  MoveL 635 to (33.53, 138.59, 49.77) mm, rotated rx 110.14 ry 0 rz -13.26 deg; joints [126.944, -22.767, 36.217, -107.187, 38.986, 156.564, 25, 13.26]
  MoveL 636 to (34.49, 138.1, 50.45) mm, rotated rx 110.14 ry 0 rz -13.26 deg; joints [126.986, -22.796, 36.22, -107.13, 39.017, 156.503, 25, 13.26]
  MoveL 637 to (34.94, 137.59, 51.53) mm, rotated rx 110.14 ry 0 rz -13.26 deg; joints [127.026, -22.799, 36.192, -107.072, 39.045, 156.439, 25, 13.26]
  MoveL 638 to (34.99, 137.43, 51.91) mm, rotated rx 110.29 ry 0 rz -13.29 deg; joints [127.07, -22.764, 36.12, -107.001, 39.075, 156.207, 25, 13.293]
  MoveL 639 to (34.9, 137.09, 52.87) mm, rotated rx 110.29 ry 0 rz -13.29 deg; joints [127.093, -22.746, 36.081, -106.964, 39.09, 156.166, 25, 13.293]
  MoveL 640 to (34.24, 136.43, 54.94) mm, rotated rx 111.13 ry 0 rz -13.09 deg; joints [127.332, -22.556, 35.689, -106.59, 39.255, 154.912, 25, 13.093]
  MoveL 641 to (34.22, 136.45, 54.91) mm, rotated rx 112.01 ry 0 rz -13.37 deg; joints [127.511, -22.368, 35.349, -106.31, 39.379, 153.728, 25, 13.374]
  MoveL 642 to (35.06, 135.89, 55.75) mm, rotated rx 112.35 ry 0 rz -13.76 deg; joints [127.61, -22.288, 35.19, -106.163, 39.45, 153.224, 25, 13.758]
  MoveL 643 to (35.03, 135.9, 55.76) mm, rotated rx 112.58 ry 0 rz -14.72 deg; joints [127.605, -22.149, 35.037, -106.15, 39.441, 152.972, 25, 14.719]
  MoveL 644 to (36.59, 135.66, 55.37) mm, rotated rx 112.43 ry 0 rz -15.36 deg; joints [127.559, -22.187, 35.111, -106.218, 39.408, 153.203, 25, 15.358]
  MoveL 645 to (37.62, 135.39, 55.32) mm, rotated rx 112.43 ry 0 rz -15.36 deg; joints [127.584, -22.23, 35.142, -106.19, 39.428, 153.175, 25, 15.358]
  MoveL 646 to (37.97, 135.27, 55.38) mm, rotated rx 112.45 ry 0 rz -15.51 deg; joints [127.591, -22.225, 35.131, -106.18, 39.433, 153.14, 25, 15.509]
  MoveL 647 to (38.54, 135.04, 55.55) mm, rotated rx 112.45 ry 0 rz -15.51 deg; joints [127.61, -22.245, 35.141, -106.156, 39.448, 153.115, 25, 15.509]
  MoveL 648 to (41.47, 133.6, 56.89) mm, rotated rx 113 ry 0 rz -16.82 deg; joints [127.768, -22.114, 34.886, -105.925, 39.562, 152.313, 25, 16.823]
  MoveL 649 to (41.44, 133.61, 56.9) mm, rotated rx 113.08 ry 0 rz -17.26 deg; joints [127.76, -22.054, 34.824, -105.927, 39.554, 152.23, 25, 17.263]
  MoveL 650 to (46.56, 131.98, 56.74) mm, rotated rx 113.02 ry 0 rz -19.47 deg; joints [127.742, -22.069, 34.854, -105.954, 39.541, 152.323, 25, 19.465]
  MoveL 651 to (46.55, 131.99, 56.74) mm, rotated rx 112.91 ry 0 rz -19.9 deg; joints [127.691, -22.047, 34.863, -106.018, 39.502, 152.499, 25, 19.901]
  MoveL 652 to (46.74, 131.96, 56.65) mm, rotated rx 112.87 ry 0 rz -19.98 deg; joints [127.68, -22.056, 34.88, -106.034, 39.494, 152.554, 25, 19.979]
  MoveL 653 to (52.44, 130.85, 54.2) mm, rotated rx 111.89 ry 0 rz -22.26 deg; joints [127.4, -22.293, 35.343, -106.454, 39.295, 153.995, 25, 22.265]
  MoveL 654 to (53.71, 130.41, 54) mm, rotated rx 111.89 ry 0 rz -22.26 deg; joints [127.427, -22.35, 35.388, -106.424, 39.317, 153.964, 25, 22.265]
  MoveL 655 to (54, 130.27, 54.04) mm, rotated rx 111.91 ry 0 rz -22.4 deg; joints [127.432, -22.347, 35.381, -106.418, 39.32, 153.943, 25, 22.396]
  MoveL 656 to (54.41, 130.07, 54.13) mm, rotated rx 111.91 ry 0 rz -22.4 deg; joints [127.445, -22.364, 35.39, -106.401, 39.33, 153.926, 25, 22.396]
  MoveL 657 to (56.76, 128.71, 54.94) mm, rotated rx 112.27 ry 0 rz -23.62 deg; joints [127.539, -22.269, 35.217, -106.258, 39.396, 153.409, 25, 23.619]
  MoveL 658 to (57.14, 128.52, 55.01) mm, rotated rx 112.29 ry 0 rz -23.79 deg; joints [127.547, -22.262, 35.204, -106.246, 39.402, 153.367, 25, 23.792]
  MoveL 659 to (60.62, 126.74, 55.41) mm, rotated rx 112.47 ry 0 rz -25.68 deg; joints [127.579, -22.192, 35.104, -106.191, 39.423, 153.132, 25, 25.675]
  MoveL 660 to (60.77, 126.66, 55.41) mm, rotated rx 112.39 ry 0 rz -26.04 deg; joints [127.544, -22.177, 35.111, -106.238, 39.397, 153.258, 25, 26.044]
  MoveL 661 to (66.75, 124.73, 52.87) mm, rotated rx 111.36 ry 0 rz -28.56 deg; joints [127.248, -22.417, 35.593, -106.687, 39.189, 154.785, 25, 28.562]
  MoveL 662 to (67.07, 124.6, 52.75) mm, rotated rx 111.21 ry 0 rz -28.89 deg; joints [127.201, -22.427, 35.638, -106.757, 39.155, 155.009, 25, 28.89]
  MoveL 663 to (71.33, 123.43, 49.83) mm, rotated rx 110.03 ry 0 rz -30.61 deg; joints [126.867, -22.688, 36.187, -107.29, 38.929, 156.774, 25, 30.614]
  MoveL 664 to (71.29, 123.43, 49.87) mm, rotated rx 109.41 ry 0 rz -31.01 deg; joints [126.706, -22.752, 36.386, -107.545, 38.819, 157.679, 25, 31.007]
  MoveL 665 to (71.98, 123.95, 47.56) mm, rotated rx 108.48 ry 0 rz -31.14 deg; joints [126.448, -22.945, 36.815, -107.982, 38.653, 159.084, 25, 31.136]
  MoveL 666 to (72.34, 124.04, 46.77) mm, rotated rx 108.48 ry 0 rz -31.14 deg; joints [126.435, -22.97, 36.853, -108.006, 38.646, 159.111, 25, 31.136]
  MoveL 667 to (72.46, 124.04, 46.59) mm, rotated rx 108.41 ry 0 rz -31.18 deg; joints [126.415, -22.984, 36.887, -108.041, 38.633, 159.221, 25, 31.175]
  MoveL 668 to (72.72, 124.02, 46.25) mm, rotated rx 108.41 ry 0 rz -31.18 deg; joints [126.413, -23, 36.907, -108.048, 38.632, 159.23, 25, 31.175]
  MoveL 669 to (73.91, 123.81, 44.88) mm, rotated rx 107.79 ry 0 rz -31.68 deg; joints [126.243, -23.116, 37.182, -108.344, 38.526, 160.175, 25, 31.678]
  MoveL 670 to (74.21, 123.77, 44.51) mm, rotated rx 107.28 ry 0 rz -31.93 deg; joints [126.117, -23.185, 37.372, -108.566, 38.447, 160.928, 25, 31.927]
  MoveL 671 to (76.55, 125.04, 36.2) mm, rotated rx 104.01 ry 0 rz -32.44 deg; joints [125.241, -23.772, 38.877, -110.247, 37.953, 166.057, 25, 32.439]
  MoveL 672 to (76.56, 125.03, 36.23) mm, rotated rx 103.38 ry 0 rz -32.31 deg; joints [125.12, -23.868, 39.115, -110.501, 37.893, 166.973, 25, 32.307]
  MoveL 673 to (75.15, 126.78, 32.95) mm, rotated rx 102.1 ry 0 rz -31.48 deg; joints [124.791, -24.064, 39.699, -111.201, 37.734, 169.031, 25, 31.478]
  MoveL 674 to (75.18, 126.76, 32.96) mm, rotated rx 101.72 ry 0 rz -31 deg; joints [124.744, -24.162, 39.871, -111.324, 37.72, 169.55, 25, 31.005]
  MoveL 675 to (72.12, 128.85, 31.65) mm, rotated rx 101.21 ry 0 rz -29.57 deg; joints [124.616, -24.235, 40.103, -111.609, 37.663, 170.376, 25, 29.568]
  MoveL 676 to (72.16, 128.83, 31.66) mm, rotated rx 101.17 ry 0 rz -29.07 deg; joints [124.64, -24.296, 40.153, -111.578, 37.681, 170.382, 25, 29.071]
  MoveL 677 to (69.26, 130.27, 32.26) mm, rotated rx 101.4 ry 0 rz -27.82 deg; joints [124.699, -24.263, 40.047, -111.448, 37.706, 170.004, 25, 27.818]
  MoveL 678 to (68.73, 130.53, 32.34) mm, rotated rx 101.43 ry 0 rz -27.65 deg; joints [124.701, -24.253, 40.032, -111.44, 37.707, 169.973, 25, 27.647]
  MoveL 679 to (65.39, 132.13, 32.76) mm, rotated rx 101.64 ry 0 rz -25.99 deg; joints [124.767, -24.248, 39.955, -111.306, 37.739, 169.608, 25, 25.986]
  MoveL 680 to (65.13, 132.23, 32.87) mm, rotated rx 101.68 ry 0 rz -25.88 deg; joints [124.777, -24.242, 39.937, -111.284, 37.744, 169.545, 25, 25.88]
  MoveL 681 to (65.15, 132.23, 32.84) mm, rotated rx 101.9 ry 0 rz -25.53 deg; joints [124.842, -24.257, 39.885, -111.156, 37.779, 169.183, 25, 25.527]
  MoveL 682 to (59.71, 133.3, 38.37) mm, rotated rx 104.07 ry 0 rz -23.42 deg; joints [125.401, -23.918, 38.899, -109.988, 38.055, 165.728, 25, 23.417]
  MoveL 683 to (58.71, 133.57, 39) mm, rotated rx 104.07 ry 0 rz -23.42 deg; joints [125.39, -23.865, 38.845, -109.994, 38.045, 165.731, 25, 23.417]
  MoveL 684 to (58.23, 133.73, 39.16) mm, rotated rx 104.13 ry 0 rz -23.22 deg; joints [125.407, -23.855, 38.816, -109.961, 38.054, 165.632, 25, 23.222]
  MoveL 685 to (57.76, 133.9, 39.27) mm, rotated rx 104.13 ry 0 rz -23.22 deg; joints [125.397, -23.832, 38.798, -109.972, 38.047, 165.644, 25, 23.222]
  MoveL 686 to (52.25, 135.95, 39.92) mm, rotated rx 104.39 ry 0 rz -20.91 deg; joints [125.465, -23.788, 38.68, -109.837, 38.083, 165.238, 25, 20.912]
  MoveL 687 to (51.7, 136.16, 39.92) mm, rotated rx 104.39 ry 0 rz -20.91 deg; joints [125.451, -23.763, 38.663, -109.857, 38.073, 165.258, 25, 20.912]
  MoveL 688 to (50.6, 136.72, 39.43) mm, rotated rx 104.39 ry 0 rz -20.91 deg; joints [125.411, -23.718, 38.647, -109.918, 38.046, 165.323, 25, 20.912]
  MoveL 689 to (50.38, 136.86, 39.24) mm, rotated rx 104.31 ry 0 rz -20.81 deg; joints [125.391, -23.731, 38.682, -109.958, 38.036, 165.444, 25, 20.811]
  MoveL 690 to (49.72, 137.39, 38.2) mm, rotated rx 104.31 ry 0 rz -20.81 deg; joints [125.349, -23.712, 38.698, -110.03, 38.01, 165.521, 25, 20.811]
  MoveL 691 to (49.04, 138.28, 35.81) mm, rotated rx 103.37 ry 0 rz -20.44 deg; joints [125.105, -23.865, 39.126, -110.529, 37.884, 167.008, 25, 20.436]
  MoveL 692 to (48.96, 138.42, 35.38) mm, rotated rx 103.37 ry 0 rz -20.44 deg; joints [125.092, -23.865, 39.139, -110.553, 37.878, 167.034, 25, 20.436]
  MoveL 693 to (49.06, 138.63, 34.37) mm, rotated rx 103.37 ry 0 rz -20.44 deg; joints [125.071, -23.879, 39.178, -110.598, 37.867, 167.084, 25, 20.436]
  MoveL 694 to (49.13, 138.66, 34.16) mm, rotated rx 103.29 ry 0 rz -20.46 deg; joints [125.05, -23.892, 39.215, -110.641, 37.857, 167.213, 25, 20.456]
  MoveL 695 to (49.47, 138.71, 33.44) mm, rotated rx 103.29 ry 0 rz -20.46 deg; joints [125.042, -23.914, 39.251, -110.663, 37.854, 167.238, 25, 20.456]
  MoveL 696 to (50.81, 138.69, 31.45) mm, rotated rx 102.52 ry 0 rz -20.95 deg; joints [124.844, -24.033, 39.603, -111.086, 37.759, 168.479, 25, 20.946]
  MoveL 697 to (51.64, 138.87, 29.25) mm, rotated rx 101.46 ry 0 rz -21.32 deg; joints [124.58, -24.168, 40.058, -111.662, 37.639, 170.18, 25, 21.317]
  MoveL 698 to (51.92, 138.88, 28.69) mm, rotated rx 101.46 ry 0 rz -21.32 deg; joints [124.574, -24.186, 40.087, -111.679, 37.638, 170.199, 25, 21.317]
  MoveL 699 to (52.11, 138.87, 28.42) mm, rotated rx 101.35 ry 0 rz -21.38 deg; joints [124.548, -24.201, 40.135, -111.738, 37.627, 170.371, 25, 21.384]
  MoveL 700 to (52.33, 138.84, 28.13) mm, rotated rx 101.35 ry 0 rz -21.38 deg; joints [124.547, -24.214, 40.152, -111.744, 37.628, 170.378, 25, 21.384]
  MoveL 701 to (53.88, 138.59, 26.37) mm, rotated rx 100.68 ry 0 rz -21.97 deg; joints [124.38, -24.304, 40.457, -112.128, 37.558, 171.479, 25, 21.975]
  MoveL 702 to (53.87, 138.59, 26.41) mm, rotated rx 100.23 ry 0 rz -22.19 deg; joints [124.281, -24.324, 40.597, -112.346, 37.516, 172.163, 25, 22.191]
  MoveL 703 to (54.09, 138.69, 25.45) mm, rotated rx 99.86 ry 0 rz -22.25 deg; joints [124.191, -24.37, 40.763, -112.559, 37.482, 172.768, 25, 22.255]
  MoveL 704 to (54.13, 138.66, 25.45) mm, rotated rx 98.75 ry 0 rz -21.31 deg; joints [124.039, -24.584, 41.228, -112.978, 37.444, 174.351, 25, 21.313]
  MoveL 705 to (46.69, 141.33, 25.56) mm, rotated rx 98.79 ry 0 rz -18.27 deg; joints [124.048, -24.58, 41.21, -112.954, 37.447, 174.284, 25, 18.27]
  MoveL 706 to (46.19, 141.5, 25.51) mm, rotated rx 98.79 ry 0 rz -18.27 deg; joints [124.034, -24.556, 41.196, -112.976, 37.439, 174.307, 25, 18.27]
  MoveL 707 to (45.76, 141.66, 25.42) mm, rotated rx 98.76 ry 0 rz -18.09 deg; joints [124.026, -24.56, 41.212, -112.997, 37.436, 174.365, 25, 18.095]
  MoveL 708 to (44.74, 142.08, 24.9) mm, rotated rx 98.76 ry 0 rz -18.09 deg; joints [123.99, -24.517, 41.199, -113.061, 37.417, 174.433, 25, 18.095]
  MoveL 709 to (41.28, 143.63, 21.8) mm, rotated rx 97.57 ry 0 rz -16.65 deg; joints [123.709, -24.645, 41.729, -113.766, 37.33, 176.407, 25, 16.645]
  MoveL 710 to (40.62, 143.96, 20.83) mm, rotated rx 97.57 ry 0 rz -16.65 deg; joints [123.674, -24.621, 41.743, -113.84, 37.314, 176.487, 25, 16.645]
  MoveL 711 to (40.51, 144.16, 19.63) mm, rotated rx 97.57 ry 0 rz -16.65 deg; joints [123.647, -24.623, 41.782, -113.905, 37.306, 176.559, 25, 16.645]
  MoveL 712 to (40.56, 144.19, 19.26) mm, rotated rx 97.43 ry 0 rz -16.66 deg; joints [123.615, -24.637, 41.844, -113.99, 37.297, 176.794, 25, 16.66]
  MoveL 713 to (40.77, 144.23, 18.53) mm, rotated rx 97.43 ry 0 rz -16.66 deg; joints [123.605, -24.651, 41.876, -114.018, 37.296, 176.826, 25, 16.66]
  MoveL 714 to (42.09, 144.19, 15.65) mm, rotated rx 96.33 ry 0 rz -17.15 deg; joints [123.355, -24.751, 42.362, -114.684, 37.237, 178.667, 25, 17.147]
  MoveL 715 to (42.15, 144.21, 15.29) mm, rotated rx 96.03 ry 0 rz -17.22 deg; joints [123.292, -24.767, 42.473, -114.851, 37.223, 179.149, 25, 17.22]
  MoveL 716 to (43.13, 144.27, 11.53) mm, rotated rx 94.6 ry 0 rz -17.57 deg; joints [122.977, -24.873, 43.099, -115.737, 37.174, 181.571, 25, 17.568]
  MoveL 717 to (43.15, 144.26, 11.55) mm, rotated rx 93.63 ry 0 rz -17.22 deg; joints [122.834, -24.962, 43.458, -116.179, 37.171, 183.042, 25, 17.224]
  MoveL 718 to (37.84, 146.01, 7.35) mm, rotated rx 92.03 ry 0 rz -15.1 deg; joints [122.503, -25.04, 44.146, -117.191, 37.164, 185.776, 25, 15.099]
  MoveL 719 to (37.83, 146.02, 7.37) mm, rotated rx 91.85 ry 0 rz -14.45 deg; joints [122.513, -25.124, 44.258, -117.214, 37.186, 185.989, 25, 14.447]
  MoveL 720 to (29.7, 147.83, 8.53) mm, rotated rx 92.3 ry 0 rz -11.23 deg; joints [122.607, -25.113, 44.071, -116.924, 37.185, 185.216, 25, 11.229]
  MoveL 721 to (28.41, 148.09, 8.36) mm, rotated rx 92.3 ry 0 rz -11.23 deg; joints [122.574, -25.052, 44.037, -116.985, 37.169, 185.279, 25, 11.229]
  MoveL 722 to (28.01, 148.18, 8.19) mm, rotated rx 92.23 ry 0 rz -11.07 deg; joints [122.561, -25.055, 44.065, -117.026, 37.169, 185.392, 25, 11.073]
  MoveL 723 to (25.31, 148.72, 6.82) mm, rotated rx 91.74 ry 0 rz -10.08 deg; joints [122.457, -25.068, 44.275, -117.351, 37.172, 186.251, 25, 10.081]
  MoveL 724 to (25.34, 148.72, 6.79) mm, rotated rx 91.84 ry 0 rz -9.07 deg; joints [122.534, -25.19, 44.323, -117.195, 37.202, 185.986, 25, 9.07]
  MoveL 725 to (23.1, 148.99, 8.62) mm, rotated rx 92.54 ry 0 rz -8.21 deg; joints [122.676, -25.161, 44.025, -116.753, 37.2, 184.791, 25, 8.214]
  MoveL 726 to (22.86, 149.01, 8.97) mm, rotated rx 92.78 ry 0 rz -8.01 deg; joints [122.728, -25.165, 43.94, -116.602, 37.204, 184.381, 25, 8.008]
  MoveL 727 to (20.3, 149.18, 11.9) mm, rotated rx 93.9 ry 0 rz -7.03 deg; joints [122.963, -25.103, 43.457, -115.9, 37.218, 182.476, 25, 7.031]
  MoveL 728 to (19.26, 149.26, 12.61) mm, rotated rx 93.9 ry 0 rz -7.03 deg; joints [122.951, -25.052, 43.401, -115.904, 37.205, 182.476, 25, 7.031]
  MoveL 729 to (18.7, 149.31, 12.81) mm, rotated rx 93.97 ry 0 rz -6.82 deg; joints [122.967, -25.048, 43.368, -115.856, 37.207, 182.347, 25, 6.817]
  MoveL 730 to (18.28, 149.35, 12.92) mm, rotated rx 93.97 ry 0 rz -6.82 deg; joints [122.96, -25.028, 43.352, -115.867, 37.202, 182.357, 25, 6.817]
  MoveL 731 to (13.22, 149.81, 13.78) mm, rotated rx 94.38 ry 0 rz -4.63 deg; joints [123.06, -25.033, 43.201, -115.597, 37.22, 181.648, 25, 4.63]
  MoveL 732 to (10.64, 149.89, 15.02) mm, rotated rx 94.86 ry 0 rz -3.65 deg; joints [123.163, -25, 42.994, -115.303, 37.234, 180.847, 25, 3.645]
  MoveL 733 to (9.93, 149.91, 15.35) mm, rotated rx 94.92 ry 0 rz -3.55 deg; joints [123.168, -24.974, 42.949, -115.274, 37.23, 180.752, 25, 3.546]
  MoveL 734 to (7.35, 149.99, 16.03) mm, rotated rx 95.18 ry 0 rz -2.56 deg; joints [123.226, -24.955, 42.835, -115.114, 37.239, 180.313, 25, 2.561]
  Set speed (16.7 mm/s)
  MoveL 735 to (8.24, 169.89, 17.83) mm, rotated rx 95.18 ry 0 rz -2.56 deg; joints [122.611, -25.564, 42.869, -114.935, 36.464, 179.857, 25, 2.561]
  Set speed (1000.0 mm/s)
  MoveL 736 to (4.59, 170.21, 15.87) mm, rotated rx 94.56 ry 0 rz -1.2 deg; joints [122.477, -25.63, 43.161, -115.325, 36.445, 180.906, 25, 1.199]
  Set speed (5.0 mm/s)
  MoveL 737 to (4.17, 150.28, 14.28) mm, rotated rx 94.56 ry 0 rz -1.2 deg; joints [123.098, -25.017, 43.119, -115.486, 37.224, 181.344, 25, 1.199]
  Set speed (16.7 mm/s)
  MoveL 738 to (2.77, 150.26, 14.91) mm, rotated rx 94.8 ry 0 rz -0.67 deg; joints [123.15, -25.001, 43.015, -115.338, 37.231, 180.939, 25, 0.665]
  MoveL 739 to (1.49, 150.25, 15.12) mm, rotated rx 94.8 ry 0 rz -0.67 deg; joints [123.124, -24.941, 42.97, -115.376, 37.215, 180.977, 25, 0.665]
  MoveL 740 to (1.28, 150.26, 15.1) mm, rotated rx 94.79 ry 0 rz -0.58 deg; joints [123.122, -24.942, 42.973, -115.381, 37.215, 180.991, 25, 0.585]
  MoveL 741 to (0.58, 150.28, 14.92) mm, rotated rx 94.79 ry 0 rz -0.58 deg; joints [123.103, -24.911, 42.959, -115.416, 37.205, 181.028, 25, 0.585]
  MoveL 742 to (-0.95, 150.34, 14.29) mm, rotated rx 94.55 ry 0 rz 0 deg; joints [123.051, -24.928, 43.063, -115.565, 37.198, 181.432, 25, 0]
  MoveL 743 to (-2.76, 150.39, 13.54) mm, rotated rx 94.27 ry 0 rz 0.69 deg; joints [122.989, -24.947, 43.187, -115.742, 37.191, 181.917, 25, -0.69]
  MoveL 744 to (-3.05, 150.39, 13.4) mm, rotated rx 94.27 ry 0 rz 0.69 deg; joints [122.98, -24.935, 43.183, -115.76, 37.187, 181.936, 25, -0.69]
  MoveL 745 to (-3.44, 150.4, 13.18) mm, rotated rx 94.18 ry 0 rz 0.84 deg; joints [122.962, -24.94, 43.22, -115.813, 37.185, 182.08, 25, -0.839]
  MoveL 746 to (-5.89, 150.44, 11.76) mm, rotated rx 93.65 ry 0 rz 1.76 deg; joints [122.847, -24.972, 43.453, -116.15, 37.174, 182.993, 25, -1.762]
  MoveL 747 to (-5.83, 150.44, 11.77) mm, rotated rx 93.52 ry 0 rz 2.26 deg; joints [122.857, -25.041, 43.537, -116.16, 37.19, 183.136, 25, -2.265]
  MoveL 748 to (-8.98, 150.28, 11.92) mm, rotated rx 93.58 ry 0 rz 3.46 deg; joints [122.869, -25.038, 43.513, -116.124, 37.191, 183.04, 25, -3.465]
  MoveL 749 to (-9.52, 150.25, 11.88) mm, rotated rx 93.58 ry 0 rz 3.46 deg; joints [122.856, -25.013, 43.498, -116.147, 37.184, 183.063, 25, -3.465]
  MoveL 750 to (-10.04, 150.22, 11.79) mm, rotated rx 93.54 ry 0 rz 3.66 deg; joints [122.849, -25.015, 43.512, -116.168, 37.183, 183.121, 25, -3.664]
  MoveL 751 to (-10.45, 150.2, 11.69) mm, rotated rx 93.54 ry 0 rz 3.66 deg; joints [122.838, -24.997, 43.504, -116.189, 37.178, 183.143, 25, -3.664]
  MoveL 752 to (-13.43, 150.04, 10.65) mm, rotated rx 93.15 ry 0 rz 4.8 deg; joints [122.754, -25.019, 43.675, -116.439, 37.174, 183.82, 25, -4.801]
  MoveL 753 to (-13.42, 150.04, 10.63) mm, rotated rx 93.18 ry 0 rz 5.52 deg; joints [122.803, -25.104, 43.721, -116.349, 37.198, 183.693, 25, -5.518]
  MoveL 754 to (-16.19, 149.67, 11.96) mm, rotated rx 93.68 ry 0 rz 6.58 deg; joints [122.909, -25.076, 43.504, -116.033, 37.204, 182.835, 25, -6.58]
  MoveL 755 to (-16.97, 149.57, 12.18) mm, rotated rx 93.68 ry 0 rz 6.58 deg; joints [122.895, -25.039, 43.472, -116.052, 37.195, 182.853, 25, -6.58]
  MoveL 756 to (-17.85, 149.46, 12.28) mm, rotated rx 93.72 ry 0 rz 6.92 deg; joints [122.903, -25.037, 43.455, -116.028, 37.195, 182.787, 25, -6.917]
  MoveL 757 to (-19.05, 149.32, 12.12) mm, rotated rx 93.72 ry 0 rz 6.92 deg; joints [122.873, -24.982, 43.425, -116.083, 37.18, 182.844, 25, -6.917]
  MoveL 758 to (-23.23, 148.85, 10.44) mm, rotated rx 93.08 ry 0 rz 8.52 deg; joints [122.738, -25.017, 43.701, -116.485, 37.172, 183.935, 25, -8.518]
  MoveL 759 to (-23.2, 148.86, 10.45) mm, rotated rx 93.07 ry 0 rz 9.16 deg; joints [122.775, -25.096, 43.757, -116.426, 37.193, 183.891, 25, -9.155]
  MoveL 760 to (-25.12, 148.5, 11.09) mm, rotated rx 93.31 ry 0 rz 9.9 deg; joints [122.826, -25.084, 43.652, -116.273, 37.195, 183.476, 25, -9.897]
  MoveL 761 to (-26.31, 148.29, 11.17) mm, rotated rx 93.2 ry 0 rz 9.91 deg; joints [122.782, -25.034, 43.652, -116.369, 37.18, 183.691, 25, -9.914]
  MoveL 762 to (-27.06, 148.18, 10.9) mm, rotated rx 93.13 ry 0 rz 9.93 deg; joints [122.748, -25.005, 43.665, -116.448, 37.17, 183.85, 25, -9.925]
  MoveL 763 to (-27.67, 148.1, 10.44) mm, rotated rx 93.06 ry 0 rz 9.94 deg; joints [122.716, -24.983, 43.687, -116.529, 37.162, 184.009, 25, -9.936]
  MoveL 764 to (-28.2, 148.05, 9.57) mm, rotated rx 92.96 ry 0 rz 9.95 deg; joints [122.674, -24.967, 43.735, -116.64, 37.155, 184.225, 25, -9.95]
  MoveL 765 to (-28.34, 148.09, 8.55) mm, rotated rx 92.87 ry 0 rz 9.96 deg; joints [122.64, -24.971, 43.799, -116.742, 37.153, 184.433, 25, -9.964]
  MoveL 766 to (-29.06, 148.04, 6.92) mm, rotated rx 92.25 ry 0 rz 10.24 deg; joints [122.512, -24.998, 44.066, -117.138, 37.154, 185.5, 25, -10.236]
  MoveL 767 to (-28.94, 148.05, 7.15) mm, rotated rx 92.25 ry 0 rz 10.24 deg; joints [122.518, -25.003, 44.061, -117.121, 37.155, 185.482, 25, -10.236]
  MoveL 768 to (-29.05, 148.04, 6.96) mm, rotated rx 92.17 ry 0 rz 10.28 deg; joints [122.503, -25.006, 44.092, -117.167, 37.156, 185.606, 25, -10.277]
  MoveL 769 to (-29.31, 148.01, 6.46) mm, rotated rx 92.03 ry 0 rz 10.35 deg; joints [122.471, -25.009, 44.157, -117.269, 37.156, 185.866, 25, -10.35]
  MoveL 770 to (-29.27, 148.01, 6.49) mm, rotated rx 91.56 ry 0 rz 10.9 deg; joints [122.431, -25.091, 44.358, -117.445, 37.178, 186.54, 25, -10.9]
  MoveL 771 to (-31.93, 147.5, 5.64) mm, rotated rx 91.23 ry 0 rz 11.93 deg; joints [122.366, -25.101, 44.496, -117.652, 37.182, 187.095, 25, -11.929]
  MoveL 772 to (-32.39, 147.41, 5.43) mm, rotated rx 91.23 ry 0 rz 11.93 deg; joints [122.352, -25.08, 44.488, -117.681, 37.177, 187.126, 25, -11.929]
  MoveL 773 to (-32.76, 147.33, 5.22) mm, rotated rx 91.15 ry 0 rz 12.07 deg; joints [122.336, -25.082, 44.522, -117.732, 37.179, 187.264, 25, -12.072]
  MoveL 774 to (-33.25, 147.24, 4.86) mm, rotated rx 91.15 ry 0 rz 12.07 deg; joints [122.319, -25.06, 44.52, -117.771, 37.174, 187.306, 25, -12.072]
  MoveL 775 to (-36.36, 146.57, 1.84) mm, rotated rx 90.01 ry 0 rz 13.28 deg; joints [122.097, -25.084, 45.002, -118.508, 37.206, 189.282, 25, -13.283]
  MoveL 776 to (-36.4, 146.55, 1.78) mm, rotated rx 89.81 ry 0 rz 13.57 deg; joints [122.083, -25.12, 45.093, -118.585, 37.22, 189.574, 25, -13.569]
  MoveL 777 to (-41.32, 145.25, -0.45) mm, rotated rx 88.96 ry 0 rz 15.5 deg; joints [121.925, -25.126, 45.446, -119.134, 37.257, 191.042, 25, -15.497]
  MoveL 778 to (-41.25, 145.28, -0.43) mm, rotated rx 88.89 ry 0 rz 15.83 deg; joints [121.936, -25.171, 45.498, -119.132, 37.27, 191.116, 25, -15.832]
  MoveL 779 to (-45.56, 143.99, -0.15) mm, rotated rx 89 ry 0 rz 17.62 deg; joints [121.961, -25.181, 45.459, -119.052, 37.267, 190.917, 25, -17.617]
  MoveL 780 to (-46.02, 143.84, -0.16) mm, rotated rx 89 ry 0 rz 17.62 deg; joints [121.95, -25.158, 45.445, -119.072, 37.262, 190.938, 25, -17.617]
  MoveL 781 to (-47.03, 143.51, -0.3) mm, rotated rx 88.95 ry 0 rz 18.02 deg; joints [121.94, -25.158, 45.467, -119.107, 37.264, 191.03, 25, -18.023]
  MoveL 782 to (-47.66, 143.3, -0.48) mm, rotated rx 88.95 ry 0 rz 18.02 deg; joints [121.922, -25.127, 45.453, -119.143, 37.258, 191.068, 25, -18.023]
  MoveL 783 to (-54.7, 140.72, -3.71) mm, rotated rx 87.72 ry 0 rz 20.87 deg; joints [121.702, -25.12, 45.959, -119.941, 37.332, 193.199, 25, -20.868]
  MoveL 784 to (-54.97, 140.61, -3.86) mm, rotated rx 87.72 ry 0 rz 20.87 deg; joints [121.693, -25.106, 45.955, -119.96, 37.33, 193.219, 25, -20.868]
  MoveL 785 to (-55.36, 140.45, -4.11) mm, rotated rx 87.62 ry 0 rz 21.03 deg; joints [121.676, -25.105, 45.994, -120.023, 37.336, 193.387, 25, -21.03]
  MoveL 786 to (-55.65, 140.33, -4.33) mm, rotated rx 87.62 ry 0 rz 21.03 deg; joints [121.666, -25.09, 45.992, -120.046, 37.335, 193.412, 25, -21.03]
  MoveL 787 to (-58.19, 139.2, -6.59) mm, rotated rx 86.76 ry 0 rz 22.09 deg; joints [121.518, -25.072, 46.343, -120.608, 37.401, 194.912, 25, -22.085]
  MoveL 788 to (-58.87, 138.86, -7.66) mm, rotated rx 86.76 ry 0 rz 22.09 deg; joints [121.487, -25.033, 46.354, -120.695, 37.402, 195.007, 25, -22.085]
  MoveL 789 to (-58.95, 138.82, -7.88) mm, rotated rx 86.68 ry 0 rz 22.12 deg; joints [121.472, -25.031, 46.389, -120.751, 37.409, 195.157, 25, -22.117]
  MoveL 790 to (-59.04, 138.76, -8.27) mm, rotated rx 86.68 ry 0 rz 22.12 deg; joints [121.465, -25.024, 46.398, -120.776, 37.411, 195.185, 25, -22.117]
  MoveL 791 to (-59.34, 138.5, -10.19) mm, rotated rx 85.95 ry 0 rz 22.26 deg; joints [121.344, -25, 46.691, -121.251, 37.479, 196.456, 25, -22.26]
  MoveL 792 to (-59.48, 138.42, -10.44) mm, rotated rx 85.61 ry 0 rz 22.4 deg; joints [121.303, -24.999, 46.812, -121.428, 37.509, 196.994, 25, -22.404]
  MoveL 793 to (-61.44, 137.13, -15.06) mm, rotated rx 83.86 ry 0 rz 23.28 deg; joints [121.031, -24.903, 47.507, -122.574, 37.714, 200.069, 25, -23.283]
  MoveL 794 to (-61.42, 137.14, -15.03) mm, rotated rx 83.46 ry 0 rz 23.66 deg; joints [121.008, -24.932, 47.66, -122.733, 37.764, 200.658, 25, -23.661]
  MoveL 795 to (-63.42, 136.09, -16.28) mm, rotated rx 82.98 ry 0 rz 24.52 deg; joints [120.939, -24.897, 47.845, -123.043, 37.83, 201.491, 25, -24.523]
  MoveL 796 to (-63.67, 135.95, -16.43) mm, rotated rx 82.92 ry 0 rz 24.64 deg; joints [120.93, -24.894, 47.87, -123.081, 37.838, 201.598, 25, -24.64]
  MoveL 797 to (-65.55, 134.9, -17.63) mm, rotated rx 82.47 ry 0 rz 25.45 deg; joints [120.866, -24.856, 48.043, -123.375, 37.905, 202.389, 25, -25.448]
  MoveL 798 to (-65.54, 134.91, -17.62) mm, rotated rx 82.36 ry 0 rz 25.99 deg; joints [120.886, -24.919, 48.122, -123.373, 37.929, 202.509, 25, -25.99]
  MoveL 799 to (-66.71, 134.35, -17.51) mm, rotated rx 82.4 ry 0 rz 26.49 deg; joints [120.891, -24.922, 48.106, -123.346, 37.922, 202.437, 25, -26.487]
  MoveL 800 to (-67.08, 134.17, -17.51) mm, rotated rx 82.4 ry 0 rz 26.49 deg; joints [120.882, -24.902, 48.093, -123.363, 37.919, 202.454, 25, -26.487]
  MoveL 801 to (-67.61, 133.9, -17.56) mm, rotated rx 82.38 ry 0 rz 26.71 deg; joints [120.879, -24.9, 48.1, -123.375, 37.922, 202.486, 25, -26.711]
  MoveL 802 to (-67.99, 133.69, -17.63) mm, rotated rx 82.38 ry 0 rz 26.71 deg; joints [120.869, -24.878, 48.088, -123.397, 37.92, 202.509, 25, -26.711]
  MoveL 803 to (-71.95, 131.43, -18.84) mm, rotated rx 81.92 ry 0 rz 28.45 deg; joints [120.806, -24.838, 48.265, -123.695, 37.991, 203.316, 25, -28.452]
  MoveL 804 to (-72.27, 131.25, -18.94) mm, rotated rx 81.88 ry 0 rz 28.58 deg; joints [120.8, -24.833, 48.278, -123.72, 37.996, 203.38, 25, -28.579]
  MoveL 805 to (-74.67, 129.78, -19.68) mm, rotated rx 81.6 ry 0 rz 29.67 deg; joints [120.763, -24.809, 48.387, -123.902, 38.043, 203.877, 25, -29.671]
  MoveL 806 to (-75.35, 129.33, -20.05) mm, rotated rx 81.6 ry 0 rz 29.67 deg; joints [120.741, -24.766, 48.373, -123.955, 38.042, 203.934, 25, -29.671]
  MoveL 807 to (-75.55, 129.19, -20.23) mm, rotated rx 81.53 ry 0 rz 29.77 deg; joints [120.732, -24.76, 48.398, -123.998, 38.053, 204.051, 25, -29.766]
  MoveL 808 to (-75.96, 128.88, -20.7) mm, rotated rx 81.53 ry 0 rz 29.77 deg; joints [120.716, -24.731, 48.397, -124.044, 38.055, 204.101, 25, -29.766]
  MoveL 809 to (-76.86, 128.09, -22.15) mm, rotated rx 80.97 ry 0 rz 30.21 deg; joints [120.643, -24.675, 48.606, -124.4, 38.15, 205.073, 25, -30.214]
  MoveL 810 to (-76.83, 128.11, -22.14) mm, rotated rx 80.62 ry 0 rz 30.97 deg; joints [120.653, -24.744, 48.773, -124.493, 38.213, 205.546, 25, -30.97]
  MoveL 811 to (-78.76, 126.95, -22.09) mm, rotated rx 80.64 ry 0 rz 31.84 deg; joints [120.655, -24.746, 48.767, -124.482, 38.209, 205.517, 25, -31.837]
  MoveL 812 to (-79.07, 126.75, -22.11) mm, rotated rx 80.64 ry 0 rz 31.84 deg; joints [120.646, -24.728, 48.756, -124.498, 38.207, 205.533, 25, -31.837]
  MoveL 813 to (-79.56, 126.43, -22.19) mm, rotated rx 80.61 ry 0 rz 32.06 deg; joints [120.643, -24.725, 48.766, -124.516, 38.212, 205.582, 25, -32.062]
  MoveL 814 to (-83.97, 123.36, -23.2) mm, rotated rx 80.21 ry 0 rz 34.26 deg; joints [120.601, -24.698, 48.926, -124.754, 38.287, 206.263, 25, -34.261]
  MoveL 815 to (-84.11, 123.27, -23.2) mm, rotated rx 80.21 ry 0 rz 34.32 deg; joints [120.602, -24.699, 48.925, -124.754, 38.287, 206.261, 25, -34.325]
  MoveL 816 to (-86.01, 122, -22.94) mm, rotated rx 80.32 ry 0 rz 35.29 deg; joints [120.619, -24.722, 48.894, -124.678, 38.269, 206.068, 25, -35.289]
  MoveL 817 to (-86.54, 121.62, -22.95) mm, rotated rx 80.32 ry 0 rz 35.29 deg; joints [120.605, -24.69, 48.874, -124.706, 38.265, 206.096, 25, -35.289]
  MoveL 818 to (-87.53, 120.87, -23.14) mm, rotated rx 80.25 ry 0 rz 35.77 deg; joints [120.596, -24.682, 48.9, -124.751, 38.278, 206.221, 25, -35.767]
  MoveL 819 to (-88.19, 120.34, -23.43) mm, rotated rx 80.25 ry 0 rz 35.77 deg; joints [120.575, -24.637, 48.882, -124.801, 38.277, 206.273, 25, -35.767]
  MoveL 820 to (-91.78, 117.05, -26.1) mm, rotated rx 79.22 ry 0 rz 37.63 deg; joints [120.452, -24.512, 49.26, -125.454, 38.475, 208.069, 25, -37.628]
  MoveL 821 to (-94.95, 113.9, -28.59) mm, rotated rx 78.17 ry 0 rz 39.59 deg; joints [120.351, -24.403, 49.655, -126.075, 38.695, 209.862, 25, -39.589]
  MoveL 822 to (-97.63, 111.54, -28.88) mm, rotated rx 78.03 ry 0 rz 41.11 deg; joints [120.345, -24.403, 49.714, -126.141, 38.726, 210.081, 25, -41.113]
  MoveL 823 to (-98.35, 110.83, -29.18) mm, rotated rx 78.03 ry 0 rz 41.11 deg; joints [120.32, -24.349, 49.69, -126.198, 38.725, 210.14, 25, -41.113]
  MoveL 824 to (-98.66, 110.49, -29.43) mm, rotated rx 77.93 ry 0 rz 41.29 deg; joints [120.31, -24.335, 49.724, -126.259, 38.747, 210.308, 25, -41.29]
  MoveL 825 to (-98.92, 110.18, -29.71) mm, rotated rx 77.93 ry 0 rz 41.29 deg; joints [120.299, -24.311, 49.719, -126.29, 38.749, 210.342, 25, -41.29]
  MoveL 826 to (-99.3, 109.59, -30.59) mm, rotated rx 77.93 ry 0 rz 41.29 deg; joints [120.277, -24.267, 49.724, -126.363, 38.762, 210.423, 25, -41.29]
  MoveL 827 to (-100.29, 106.94, -36.23) mm, rotated rx 75.74 ry 0 rz 42.26 deg; joints [120.066, -23.905, 50.488, -127.705, 39.289, 214.224, 25, -42.264]
  MoveL 828 to (-100.26, 106.61, -37.26) mm, rotated rx 75.74 ry 0 rz 42.26 deg; joints [120.054, -23.879, 50.511, -127.765, 39.31, 214.295, 25, -42.264]
  MoveL 829 to (-99.99, 106.37, -38.65) mm, rotated rx 75.2 ry 0 rz 42.25 deg; joints [120.008, -23.778, 50.694, -128.091, 39.453, 215.232, 25, -42.247]
  MoveL 830 to (-99.85, 106.32, -39.13) mm, rotated rx 75.2 ry 0 rz 42.25 deg; joints [120.006, -23.773, 50.71, -128.113, 39.464, 215.259, 25, -42.247]
  MoveL 831 to (-99.3, 106.47, -40.12) mm, rotated rx 75.2 ry 0 rz 42.25 deg; joints [120.01, -23.783, 50.755, -128.141, 39.489, 215.298, 25, -42.247]
  MoveL 832 to (-95.86, 107.97, -44.27) mm, rotated rx 73.55 ry 0 rz 40.83 deg; joints [119.886, -23.446, 51.297, -129.108, 39.952, 218.127, 25, -40.834]
  MoveL 833 to (-92.33, 109.27, -48.4) mm, rotated rx 71.91 ry 0 rz 39.42 deg; joints [119.784, -23.068, 51.82, -130.045, 40.456, 220.937, 25, -39.421]
  MoveL 834 to (-90.69, 109.58, -50.75) mm, rotated rx 70.84 ry 0 rz 38.74 deg; joints [119.726, -22.797, 52.132, -130.63, 40.795, 222.735, 25, -38.744]
  MoveL 835 to (-90.15, 109.74, -51.35) mm, rotated rx 70.54 ry 0 rz 38.5 deg; joints [119.711, -22.717, 52.216, -130.791, 40.892, 223.24, 25, -38.498]
  MoveL 836 to (-87.46, 109.87, -55.55) mm, rotated rx 68.83 ry 0 rz 37.6 deg; joints [119.647, -22.246, 52.717, -131.701, 41.491, 226.115, 25, -37.604]
  MoveL 837 to (-87.46, 109.88, -55.52) mm, rotated rx 68.22 ry 0 rz 37.52 deg; joints [119.629, -22.096, 52.847, -131.956, 41.666, 227.057, 25, -37.525]
  MoveL 838 to (-87.35, 108.92, -57.57) mm, rotated rx 67.38 ry 0 rz 37.73 deg; joints [119.609, -21.842, 53.08, -132.383, 41.981, 228.452, 25, -37.728]
  MoveL 839 to (-87.26, 108.71, -58.1) mm, rotated rx 67.38 ry 0 rz 37.73 deg; joints [119.607, -21.825, 53.091, -132.408, 41.998, 228.485, 25, -37.728]
  MoveL 840 to (-87.16, 108.58, -58.48) mm, rotated rx 67.22 ry 0 rz 37.73 deg; joints [119.604, -21.775, 53.134, -132.488, 42.059, 228.749, 25, -37.726]
  MoveL 841 to (-87.08, 108.51, -58.74) mm, rotated rx 67.22 ry 0 rz 37.73 deg; joints [119.604, -21.769, 53.141, -132.498, 42.068, 228.763, 25, -37.726]
  MoveL 842 to (-85.74, 107.56, -62.34) mm, rotated rx 65.73 ry 0 rz 37.52 deg; joints [119.586, -21.285, 53.538, -133.227, 42.656, 231.229, 25, -37.524]
  MoveL 843 to (-85.5, 107.47, -62.83) mm, rotated rx 65.73 ry 0 rz 37.52 deg; joints [119.588, -21.277, 53.554, -133.243, 42.674, 231.253, 25, -37.524]
  MoveL 844 to (-85.36, 107.44, -63.08) mm, rotated rx 65.63 ry 0 rz 37.48 deg; joints [119.588, -21.242, 53.58, -133.293, 42.716, 231.423, 25, -37.484]
  MoveL 845 to (-85.15, 107.42, -63.39) mm, rotated rx 65.63 ry 0 rz 37.48 deg; joints [119.591, -21.24, 53.593, -133.3, 42.727, 231.436, 25, -37.484]
  MoveL 846 to (-84.01, 107.4, -64.91) mm, rotated rx 64.99 ry 0 rz 37.11 deg; joints [119.59, -21.019, 53.756, -133.601, 42.991, 232.488, 25, -37.108]
  MoveL 847 to (-84.04, 107.41, -64.86) mm, rotated rx 64.47 ry 0 rz 36.99 deg; joints [119.585, -20.864, 53.847, -133.798, 43.158, 233.268, 25, -36.993]
  MoveL 848 to (-83.77, 106.83, -66.17) mm, rotated rx 63.92 ry 0 rz 37.05 deg; joints [119.588, -20.666, 53.982, -134.048, 43.391, 234.166, 25, -37.051]
  MoveL 849 to (-83.49, 106.57, -66.94) mm, rotated rx 63.92 ry 0 rz 37.05 deg; joints [119.59, -20.644, 54.001, -134.077, 43.42, 234.206, 25, -37.051]
  MoveL 850 to (-83.37, 106.52, -67.16) mm, rotated rx 63.82 ry 0 rz 37.02 deg; joints [119.591, -20.609, 54.024, -134.12, 43.461, 234.362, 25, -37.024]
  MoveL 851 to (-82.97, 106.45, -67.77) mm, rotated rx 63.82 ry 0 rz 37.02 deg; joints [119.598, -20.604, 54.047, -134.134, 43.485, 234.386, 25, -37.024]
  MoveL 852 to (-80.87, 106.44, -70.28) mm, rotated rx 62.75 ry 0 rz 36.31 deg; joints [119.614, -20.201, 54.299, -134.605, 43.953, 236.125, 25, -36.305]
  MoveL 853 to (-80.38, 106.41, -70.87) mm, rotated rx 62.47 ry 0 rz 36.13 deg; joints [119.618, -20.094, 54.361, -134.723, 44.074, 236.569, 25, -36.13]
  MoveL 854 to (-80.11, 106.42, -71.17) mm, rotated rx 62.47 ry 0 rz 36.13 deg; joints [119.624, -20.095, 54.375, -134.727, 44.086, 236.578, 25, -36.13]
  MoveL 855 to (-75.14, 106.77, -75.91) mm, rotated rx 60.41 ry 0 rz 34.27 deg; joints [119.686, -19.261, 54.823, -135.572, 45.031, 239.88, 25, -34.274]
  MoveL 856 to (-74.77, 106.81, -76.21) mm, rotated rx 60.41 ry 0 rz 34.27 deg; joints [119.694, -19.267, 54.841, -135.572, 45.045, 239.886, 25, -34.274]
  MoveL 857 to (-73.82, 107.15, -76.66) mm, rotated rx 60.41 ry 0 rz 34.27 deg; joints [119.717, -19.298, 54.884, -135.553, 45.066, 239.879, 25, -34.274]
  MoveL 858 to (-73.35, 107.38, -76.79) mm, rotated rx 60.35 ry 0 rz 34.04 deg; joints [119.719, -19.275, 54.895, -135.575, 45.092, 239.966, 25, -34.043]
  MoveL 859 to (-73.05, 107.55, -76.85) mm, rotated rx 60.35 ry 0 rz 34.04 deg; joints [119.727, -19.29, 54.908, -135.565, 45.095, 239.958, 25, -34.043]
  MoveL 860 to (-68.65, 110, -77.42) mm, rotated rx 60.1 ry 0 rz 31.82 deg; joints [119.737, -19.184, 54.96, -135.663, 45.214, 240.357, 25, -31.824]
  MoveL 861 to (-66.58, 110.63, -78.32) mm, rotated rx 59.61 ry 0 rz 30.55 deg; joints [119.741, -18.941, 55.027, -135.872, 45.438, 241.15, 25, -30.55]
  MoveL 862 to (-65.98, 110.84, -78.54) mm, rotated rx 59.42 ry 0 rz 30.09 deg; joints [119.74, -18.846, 55.046, -135.951, 45.519, 241.454, 25, -30.095]
  MoveL 863 to (-60.49, 111.53, -81.89) mm, rotated rx 57.91 ry 0 rz 27.79 deg; joints [119.82, -18.174, 55.329, -136.499, 46.253, 243.815, 25, -27.785]
  MoveL 864 to (-60.48, 111.53, -81.9) mm, rotated rx 57.06 ry 0 rz 27.35 deg; joints [119.841, -17.815, 55.413, -136.765, 46.586, 245.07, 25, -27.347]
  MoveL 865 to (-59.61, 108.8, -86.12) mm, rotated rx 55.14 ry 0 rz 27.57 deg; joints [119.98, -16.891, 55.726, -137.388, 47.567, 248.036, 25, -27.571]
  MoveL 866 to (-59.48, 108.55, -86.53) mm, rotated rx 55.14 ry 0 rz 27.57 deg; joints [119.983, -16.871, 55.732, -137.4, 47.588, 248.057, 25, -27.571]
  MoveL 867 to (-58.88, 108.18, -87.39) mm, rotated rx 55.14 ry 0 rz 27.57 deg; joints [119.998, -16.847, 55.758, -137.415, 47.633, 248.092, 25, -27.571]
  MoveL 868 to (-58.7, 108.13, -87.58) mm, rotated rx 55.05 ry 0 rz 27.51 deg; joints [120.005, -16.803, 55.771, -137.441, 47.678, 248.225, 25, -27.506]
  MoveL 869 to (-58.54, 108.09, -87.73) mm, rotated rx 55.05 ry 0 rz 27.51 deg; joints [120.009, -16.802, 55.778, -137.442, 47.686, 248.229, 25, -27.506]
  MoveL 870 to (-56.56, 107.72, -89.47) mm, rotated rx 54.23 ry 0 rz 26.76 deg; joints [120.078, -16.391, 55.897, -137.685, 48.113, 249.475, 25, -26.758]
  MoveL 871 to (-54.65, 107.13, -91.35) mm, rotated rx 53.27 ry 0 rz 26.01 deg; joints [120.162, -15.899, 56.02, -137.956, 48.612, 250.924, 25, -26.014]
  MoveL 872 to (-54.31, 107.05, -91.64) mm, rotated rx 53.27 ry 0 rz 26.01 deg; joints [120.171, -15.897, 56.034, -137.955, 48.629, 250.931, 25, -26.014]
  MoveL 873 to (-53.99, 107.01, -91.88) mm, rotated rx 53.16 ry 0 rz 25.89 deg; joints [120.182, -15.837, 56.049, -137.987, 48.69, 251.103, 25, -25.885]
  MoveL 874 to (-51.7, 106.68, -93.55) mm, rotated rx 52.36 ry 0 rz 24.96 deg; joints [120.262, -15.414, 56.148, -138.199, 49.119, 252.306, 25, -24.963]
  MoveL 875 to (-51.72, 106.71, -93.51) mm, rotated rx 51.87 ry 0 rz 24.67 deg; joints [120.288, -15.178, 56.17, -138.317, 49.325, 253.004, 25, -24.665]
  MoveL 876 to (-51.32, 106.17, -94.35) mm, rotated rx 51.46 ry 0 rz 24.59 deg; joints [120.332, -14.959, 56.216, -138.418, 49.544, 253.608, 25, -24.593]
  MoveL 877 to (-51.01, 105.9, -94.82) mm, rotated rx 51.46 ry 0 rz 24.59 deg; joints [120.34, -14.941, 56.227, -138.425, 49.571, 253.627, 25, -24.593]
  MoveL 878 to (-50.61, 105.7, -95.25) mm, rotated rx 51.43 ry 0 rz 24.58 deg; joints [120.354, -14.914, 56.244, -138.435, 49.61, 253.689, 25, -24.575]
  MoveL 879 to (-49.82, 105.45, -95.95) mm, rotated rx 51.09 ry 0 rz 24.27 deg; joints [120.392, -14.726, 56.281, -138.518, 49.797, 254.2, 25, -24.274]
  MoveL 880 to (-49.34, 104.96, -96.73) mm, rotated rx 50.4 ry 0 rz 23.98 deg; joints [120.456, -14.363, 56.331, -138.675, 50.139, 255.199, 25, -23.981]
  MoveL 881 to (-49.02, 104.73, -97.14) mm, rotated rx 50.4 ry 0 rz 23.98 deg; joints [120.465, -14.349, 56.343, -138.678, 50.163, 255.214, 25, -23.981]
  MoveL 882 to (-48.71, 104.57, -97.47) mm, rotated rx 50.23 ry 0 rz 23.87 deg; joints [120.484, -14.257, 56.358, -138.715, 50.253, 255.457, 25, -23.871]
  MoveL 883 to (-48.28, 104.42, -97.85) mm, rotated rx 50.23 ry 0 rz 23.87 deg; joints [120.496, -14.251, 56.374, -138.714, 50.275, 255.467, 25, -23.871]
  MoveL 884 to (-43.98, 103.32, -100.99) mm, rotated rx 48.64 ry 0 rz 22.09 deg; joints [120.695, -13.344, 56.51, -139.051, 51.157, 257.804, 25, -22.086]
  MoveL 885 to (-43.55, 103.24, -101.26) mm, rotated rx 48.64 ry 0 rz 22.09 deg; joints [120.707, -13.345, 56.526, -139.045, 51.174, 257.808, 25, -22.086]
  MoveL 886 to (-42.45, 103.34, -101.62) mm, rotated rx 48.64 ry 0 rz 22.09 deg; joints [120.735, -13.373, 56.568, -139.02, 51.199, 257.8, 25, -22.086]
  MoveL 887 to (-41.64, 103.55, -101.74) mm, rotated rx 48.58 ry 0 rz 21.66 deg; joints [120.744, -13.337, 56.573, -139.033, 51.233, 257.891, 25, -21.662]
  MoveL 888 to (-40.85, 103.85, -101.76) mm, rotated rx 48.58 ry 0 rz 21.66 deg; joints [120.763, -13.376, 56.604, -139.007, 51.236, 257.87, 25, -21.662]
  MoveL 889 to (-39.94, 104.31, -101.64) mm, rotated rx 48.64 ry 0 rz 21.14 deg; joints [120.755, -13.41, 56.6, -138.995, 51.204, 257.785, 25, -21.141]
  MoveL 890 to (-39.97, 104.32, -101.62) mm, rotated rx 47.2 ry 0 rz 19.88 deg; joints [120.853, -12.63, 56.586, -139.284, 51.83, 259.792, 25, -19.877]
  MoveL 891 to (-40.46, 103.11, -102.66) mm, rotated rx 46.67 ry 0 rz 20.33 deg; joints [120.928, -12.313, 56.617, -139.377, 52.129, 260.558, 25, -20.325]
  MoveL 892 to (-40.5, 102.15, -103.6) mm, rotated rx 46.67 ry 0 rz 20.33 deg; joints [120.934, -12.233, 56.609, -139.406, 52.186, 260.613, 25, -20.325]
  MoveL 893 to (-40.38, 101.81, -103.97) mm, rotated rx 46.47 ry 0 rz 20.33 deg; joints [120.963, -12.116, 56.62, -139.438, 52.297, 260.895, 25, -20.328]
  MoveL 894 to (-39.8, 101.13, -104.86) mm, rotated rx 46.47 ry 0 rz 20.33 deg; joints [120.984, -12.071, 56.636, -139.446, 52.354, 260.931, 25, -20.328]
  MoveL 895 to (-37.19, 99.47, -107.37) mm, rotated rx 45.13 ry 0 rz 19.31 deg; joints [121.187, -11.25, 56.695, -139.653, 53.116, 262.858, 25, -19.311]
  MoveL 896 to (-36.15, 99.14, -108.04) mm, rotated rx 45.13 ry 0 rz 19.31 deg; joints [121.218, -11.244, 56.73, -139.638, 53.161, 262.871, 25, -19.311]
  MoveL 897 to (-35.88, 99.12, -108.15) mm, rotated rx 45.07 ry 0 rz 19.18 deg; joints [121.228, -11.207, 56.732, -139.646, 53.195, 262.956, 25, -19.177]
  MoveL 898 to (-35.2, 99.14, -108.35) mm, rotated rx 45.07 ry 0 rz 19.18 deg; joints [121.246, -11.223, 56.757, -139.631, 53.211, 262.952, 25, -19.177]
  MoveL 899 to (-31.81, 99.55, -109.02) mm, rotated rx 44.7 ry 0 rz 17.35 deg; joints [121.304, -10.996, 56.768, -139.681, 53.418, 263.47, 25, -17.346]
  MoveL 900 to (-31.5, 99.6, -109.07) mm, rotated rx 44.7 ry 0 rz 17.35 deg; joints [121.312, -11.007, 56.78, -139.673, 53.422, 263.466, 25, -17.346]
  MoveL 901 to (-31.19, 99.66, -109.1) mm, rotated rx 44.68 ry 0 rz 17.17 deg; joints [121.315, -10.996, 56.781, -139.675, 53.432, 263.492, 25, -17.174]
  MoveL 902 to (-29.78, 99.83, -109.33) mm, rotated rx 44.54 ry 0 rz 16.3 deg; joints [121.333, -10.9, 56.777, -139.699, 53.511, 263.696, 25, -16.302]
  MoveL 903 to (-29.79, 99.83, -109.32) mm, rotated rx 43.61 ry 0 rz 15.24 deg; joints [121.41, -10.351, 56.722, -139.848, 53.923, 264.976, 25, -15.24]
  MoveL 904 to (-29.36, 98.21, -110.91) mm, rotated rx 42.73 ry 0 rz 15.25 deg; joints [121.557, -9.797, 56.734, -139.948, 54.421, 266.206, 25, -15.247]
  MoveL 905 to (-29.24, 97.91, -111.2) mm, rotated rx 42.73 ry 0 rz 15.25 deg; joints [121.564, -9.776, 56.736, -139.951, 54.441, 266.22, 25, -15.247]
  MoveL 906 to (-28.73, 97.35, -111.82) mm, rotated rx 42.73 ry 0 rz 15.25 deg; joints [121.585, -9.745, 56.75, -139.949, 54.485, 266.242, 25, -15.247]
  MoveL 907 to (-28.33, 97.08, -112.16) mm, rotated rx 42.54 ry 0 rz 15.07 deg; joints [121.617, -9.624, 56.751, -139.969, 54.592, 266.506, 25, -15.071]
  Set speed (16.7 mm/s)
  MoveL 908 to (-31.85, 110.14, -126.89) mm, rotated rx 42.54 ry 0 rz 15.07 deg; joints [120.937, -9.792, 57.246, -140.87, 54.55, 267.198, 25, -15.071]
  Set speed (1000.0 mm/s)
  MoveL 909 to (-30.55, 107.92, -129.11) mm, rotated rx 41.19 ry 0 rz 14.57 deg; joints [121.171, -8.909, 57.23, -140.994, 55.323, 269.072, 25, -14.57]
  Set speed (5.0 mm/s)
  MoveL 910 to (-27.24, 95.17, -114.05) mm, rotated rx 41.19 ry 0 rz 14.57 deg; joints [121.841, -8.775, 56.736, -140.098, 55.329, 268.374, 25, -14.57]
  Set speed (16.7 mm/s)
  MoveL 911 to (-27.07, 94.92, -114.3) mm, rotated rx 41.04 ry 0 rz 14.51 deg; joints [121.868, -8.681, 56.734, -140.11, 55.411, 268.576, 25, -14.513]
  MoveL 912 to (-26.62, 94.47, -114.78) mm, rotated rx 41.04 ry 0 rz 14.51 deg; joints [121.886, -8.657, 56.746, -140.106, 55.446, 268.592, 25, -14.513]
  MoveL 913 to (-25.14, 93.4, -115.97) mm, rotated rx 40.33 ry 0 rz 13.81 deg; joints [122.017, -8.194, 56.733, -140.159, 55.848, 269.57, 25, -13.814]
  MoveL 914 to (-25.15, 93.43, -115.95) mm, rotated rx 39.74 ry 0 rz 13.59 deg; joints [122.096, -7.874, 56.708, -140.201, 56.108, 270.34, 25, -13.594]
  MoveL 915 to (-25.01, 92.14, -117.01) mm, rotated rx 39.11 ry 0 rz 13.69 deg; joints [122.217, -7.458, 56.689, -140.238, 56.464, 271.202, 25, -13.69]
  MoveL 916 to (-24.75, 91.45, -117.61) mm, rotated rx 39.11 ry 0 rz 13.69 deg; joints [122.234, -7.411, 56.69, -140.239, 56.507, 271.228, 25, -13.69]
  MoveL 917 to (-24.52, 91.12, -117.91) mm, rotated rx 38.93 ry 0 rz 13.6 deg; joints [122.27, -7.288, 56.683, -140.249, 56.611, 271.48, 25, -13.605]
  MoveL 918 to (-24, 90.62, -118.4) mm, rotated rx 38.93 ry 0 rz 13.6 deg; joints [122.291, -7.263, 56.695, -140.242, 56.649, 271.496, 25, -13.605]
  MoveL 919 to (-22.5, 89.61, -119.46) mm, rotated rx 38.27 ry 0 rz 12.84 deg; joints [122.421, -6.826, 56.667, -140.271, 57.017, 272.388, 25, -12.836]
  MoveL 920 to (-22.5, 89.65, -119.43) mm, rotated rx 37.03 ry 0 rz 13.05 deg; joints [122.628, -6.188, 56.631, -140.294, 57.564, 273.965, 25, -13.054]
  MoveL 921 to (-24.87, 86.81, -121.05) mm, rotated rx 36.02 ry 0 rz 14.91 deg; joints [122.838, -5.507, 56.567, -140.315, 58.125, 275.317, 25, -14.909]
  MoveL 922 to (-25.28, 85.96, -121.57) mm, rotated rx 36.02 ry 0 rz 14.91 deg; joints [122.839, -5.432, 56.539, -140.333, 58.161, 275.352, 25, -14.909]
  MoveL 923 to (-25.23, 85.07, -122.2) mm, rotated rx 36.02 ry 0 rz 14.91 deg; joints [122.854, -5.366, 56.526, -140.338, 58.208, 275.384, 25, -14.909]
  MoveL 924 to (-25.12, 84.72, -122.47) mm, rotated rx 35.85 ry 0 rz 14.89 deg; joints [122.891, -5.247, 56.514, -140.34, 58.304, 275.617, 25, -14.894]
  MoveL 925 to (-24.62, 83.97, -123.09) mm, rotated rx 35.85 ry 0 rz 14.89 deg; joints [122.916, -5.202, 56.518, -140.333, 58.353, 275.641, 25, -14.894]
  MoveL 926 to (-22.9, 82.39, -124.47) mm, rotated rx 34.92 ry 0 rz 14.05 deg; joints [123.117, -4.57, 56.445, -140.334, 58.863, 276.875, 25, -14.051]
  MoveL 927 to (-22.92, 82.41, -124.46) mm, rotated rx 34.46 ry 0 rz 13.87 deg; joints [123.189, -4.315, 56.404, -140.339, 59.056, 277.45, 25, -13.871]
  MoveL 928 to (-22.74, 81.54, -125.06) mm, rotated rx 34.05 ry 0 rz 13.89 deg; joints [123.28, -4.036, 56.368, -140.334, 59.278, 277.988, 25, -13.894]
  MoveL 929 to (-22.54, 81.02, -125.44) mm, rotated rx 34.05 ry 0 rz 13.89 deg; joints [123.294, -4.002, 56.365, -140.331, 59.308, 278.004, 25, -13.894]
  MoveL 930 to (-22.42, 80.81, -125.59) mm, rotated rx 33.95 ry 0 rz 13.85 deg; joints [123.318, -3.929, 56.355, -140.329, 59.366, 278.144, 25, -13.848]
  MoveL 931 to (-22.2, 80.51, -125.83) mm, rotated rx 33.95 ry 0 rz 13.85 deg; joints [123.329, -3.912, 56.357, -140.325, 59.385, 278.152, 25, -13.848]
  MoveL 932 to (-21.5, 79.72, -126.44) mm, rotated rx 33.51 ry 0 rz 13.51 deg; joints [123.426, -3.616, 56.315, -140.316, 59.618, 278.72, 25, -13.507]
  MoveL 933 to (-21.49, 79.74, -126.44) mm, rotated rx 32.68 ry 0 rz 13.58 deg; joints [123.58, -3.168, 56.252, -140.295, 59.973, 279.76, 25, -13.576]
  MoveL 934 to (-22.41, 77.11, -127.9) mm, rotated rx 31.66 ry 0 rz 14.64 deg; joints [123.817, -2.464, 56.136, -140.257, 60.516, 281.087, 25, -14.636]
  MoveL 935 to (-22.43, 77.01, -127.96) mm, rotated rx 31.53 ry 0 rz 14.78 deg; joints [123.847, -2.394, 56.129, -140.248, 60.575, 281.246, 25, -14.779]
  MoveL 936 to (-23.67, 74.16, -129.41) mm, rotated rx 30.49 ry 0 rz 16.19 deg; joints [124.096, -1.673, 55.998, -140.194, 61.123, 282.592, 25, -16.186]
  MoveL 937 to (-23.69, 74.17, -129.4) mm, rotated rx 30.27 ry 0 rz 16.63 deg; joints [124.151, -1.578, 55.997, -140.17, 61.215, 282.851, 25, -16.629]
  MoveL 938 to (-26.22, 70.97, -130.7) mm, rotated rx 29.31 ry 0 rz 19.11 deg; joints [124.384, -0.913, 55.863, -140.108, 61.709, 284.075, 25, -19.111]
  Set speed (16.7 mm/s)
  MoveL 939 to (-29.43, 80.22, -148.14) mm, rotated rx 29.31 ry 0 rz 19.11 deg; joints [123.822, -0.736, 56.313, -140.915, 61.99, 284.807, 25, -19.111]
  Set speed (1000.0 mm/s)
  MoveL 940 to (-28.39, 76.79, -150.15) mm, rotated rx 29.19 ry 0 rz 19.06 deg; joints [123.925, -0.428, 56.242, -140.885, 62.21, 285.05, 25, -19.061]
  Set speed (5.0 mm/s)
  MoveL 941 to (-25.2, 67.57, -132.69) mm, rotated rx 29.19 ry 0 rz 19.06 deg; joints [124.484, -0.61, 55.793, -140.082, 61.925, 284.319, 25, -19.061]
  Set speed (16.7 mm/s)
  MoveL 942 to (-23.44, 66.82, -133.39) mm, rotated rx 28.62 ry 0 rz 17.89 deg; joints [124.625, -0.219, 55.708, -140.038, 62.211, 285.038, 25, -17.888]
  MoveL 943 to (-22.89, 66.66, -133.57) mm, rotated rx 28.62 ry 0 rz 17.89 deg; joints [124.644, -0.216, 55.721, -140.024, 62.23, 285.04, 25, -17.888]
  MoveL 944 to (-21.54, 66.75, -133.74) mm, rotated rx 28.62 ry 0 rz 17.89 deg; joints [124.682, -0.243, 55.764, -139.989, 62.256, 285.033, 25, -17.888]
  MoveL 945 to (-21.39, 66.8, -133.74) mm, rotated rx 28.62 ry 0 rz 17.75 deg; joints [124.682, -0.243, 55.764, -139.989, 62.256, 285.033, 25, -17.752]
  MoveL 946 to (-21.09, 66.94, -133.72) mm, rotated rx 28.64 ry 0 rz 17.39 deg; joints [124.675, -0.25, 55.762, -139.993, 62.246, 285.014, 25, -17.386]
  MoveL 947 to (-20.32, 67.13, -133.74) mm, rotated rx 28.62 ry 0 rz 16.74 deg; joints [124.679, -0.239, 55.76, -139.992, 62.255, 285.034, 25, -16.742]
  MoveL 948 to (-19.09, 67.49, -133.74) mm, rotated rx 28.62 ry 0 rz 15.8 deg; joints [124.682, -0.244, 55.764, -139.989, 62.256, 285.033, 25, -15.796]
  MoveL 949 to (-18.33, 67.84, -133.67) mm, rotated rx 28.67 ry 0 rz 15.66 deg; joints [124.685, -0.302, 55.796, -139.976, 62.236, 284.964, 25, -15.656]
  MoveL 950 to (-17.72, 68.39, -133.48) mm, rotated rx 28.72 ry 0 rz 15.52 deg; joints [124.681, -0.372, 55.827, -139.968, 62.205, 284.891, 25, -15.517]
  MoveL 951 to (-14.72, 70.88, -132.54) mm, rotated rx 29.47 ry 0 rz 12.68 deg; joints [124.492, -0.894, 55.939, -140.027, 61.822, 283.93, 25, -12.679]
  MoveL 952 to (-14.46, 71.1, -132.45) mm, rotated rx 29.51 ry 0 rz 12.56 deg; joints [124.484, -0.93, 55.951, -140.027, 61.8, 283.878, 25, -12.558]
  MoveL 953 to (-14.22, 71.35, -132.34) mm, rotated rx 29.51 ry 0 rz 12.56 deg; joints [124.487, -0.954, 55.964, -140.021, 61.793, 283.87, 25, -12.558]
  MoveL 954 to (-13.06, 72.66, -131.75) mm, rotated rx 29.98 ry 0 rz 11.44 deg; joints [124.37, -1.278, 56.03, -140.054, 61.552, 283.268, 25, -11.443]
  MoveL 955 to (-12.27, 73.21, -131.52) mm, rotated rx 30.27 ry 0 rz 10.44 deg; joints [124.295, -1.448, 56.051, -140.081, 61.411, 282.908, 25, -10.441]
  MoveL 956 to (-11.79, 73.66, -131.31) mm, rotated rx 30.27 ry 0 rz 10.44 deg; joints [124.3, -1.491, 56.076, -140.07, 61.398, 282.892, 25, -10.441]
  MoveL 957 to (-11.6, 73.89, -131.2) mm, rotated rx 30.36 ry 0 rz 10.26 deg; joints [124.279, -1.552, 56.088, -140.075, 61.353, 282.78, 25, -10.263]
  MoveL 958 to (-11.34, 74.28, -131) mm, rotated rx 30.36 ry 0 rz 10.26 deg; joints [124.279, -1.586, 56.104, -140.069, 61.339, 282.766, 25, -10.263]
  MoveL 959 to (-9.75, 77.15, -129.46) mm, rotated rx 31.52 ry 0 rz 8.71 deg; joints [123.998, -2.391, 56.252, -140.133, 60.73, 281.264, 25, -8.714]
  MoveL 960 to (-8.68, 78.06, -128.99) mm, rotated rx 32.08 ry 0 rz 7.46 deg; joints [123.864, -2.726, 56.294, -140.169, 60.454, 280.559, 25, -7.464]
  MoveL 961 to (-8.12, 78.78, -128.59) mm, rotated rx 32.08 ry 0 rz 7.46 deg; joints [123.865, -2.794, 56.325, -140.155, 60.426, 280.532, 25, -7.464]
  MoveL 962 to (-8.05, 78.92, -128.51) mm, rotated rx 32.14 ry 0 rz 7.4 deg; joints [123.851, -2.836, 56.332, -140.157, 60.394, 280.453, 25, -7.4]
  MoveL 963 to (-7.91, 79.29, -128.29) mm, rotated rx 32.14 ry 0 rz 7.4 deg; joints [123.848, -2.866, 56.343, -140.154, 60.378, 280.441, 25, -7.4]
  MoveL 964 to (-7.49, 80.82, -127.35) mm, rotated rx 32.81 ry 0 rz 6.96 deg; joints [123.692, -3.328, 56.417, -140.177, 60.02, 279.567, 25, -6.964]
  MoveL 965 to (-6.64, 82.04, -126.62) mm, rotated rx 33.57 ry 0 rz 6.04 deg; joints [123.522, -3.803, 56.478, -140.205, 59.636, 278.592, 25, -6.037]
  MoveL 966 to (-6.48, 82.31, -126.45) mm, rotated rx 33.57 ry 0 rz 6.04 deg; joints [123.52, -3.827, 56.487, -140.201, 59.624, 278.581, 25, -6.037]
  MoveL 967 to (-6.28, 82.72, -126.19) mm, rotated rx 33.75 ry 0 rz 5.86 deg; joints [123.479, -3.952, 56.505, -140.204, 59.526, 278.342, 25, -5.865]
  MoveL 968 to (-6.17, 82.97, -126.04) mm, rotated rx 33.75 ry 0 rz 5.86 deg; joints [123.477, -3.973, 56.511, -140.201, 59.514, 278.333, 25, -5.865]
  MoveL 969 to (-4.86, 86.58, -123.64) mm, rotated rx 35.38 ry 0 rz 4.75 deg; joints [123.116, -5.088, 56.653, -140.215, 58.624, 276.177, 25, -4.753]
  MoveL 970 to (-4.77, 87.47, -123.02) mm, rotated rx 35.38 ry 0 rz 4.75 deg; joints [123.101, -5.154, 56.667, -140.21, 58.577, 276.145, 25, -4.753]
  MoveL 971 to (-4.81, 87.73, -122.83) mm, rotated rx 35.51 ry 0 rz 4.77 deg; joints [123.074, -5.239, 56.676, -140.21, 58.509, 275.98, 25, -4.766]
  MoveL 972 to (-4.87, 87.98, -122.65) mm, rotated rx 35.51 ry 0 rz 4.77 deg; joints [123.068, -5.255, 56.677, -140.211, 58.495, 275.972, 25, -4.766]
  MoveL 973 to (-5.21, 89.02, -121.87) mm, rotated rx 36 ry 0 rz 4.93 deg; joints [122.961, -5.593, 56.712, -140.206, 58.22, 275.309, 25, -4.929]
  MoveL 974 to (-5.24, 89.01, -121.88) mm, rotated rx 36.91 ry 0 rz 4.4 deg; joints [122.791, -6.042, 56.728, -140.217, 57.818, 274.173, 25, -4.404]
  MoveL 975 to (-4.26, 89.78, -121.36) mm, rotated rx 37.25 ry 0 rz 3.74 deg; joints [122.72, -6.269, 56.748, -140.209, 57.63, 273.72, 25, -3.737]
  MoveL 976 to (-3.87, 90.15, -121.1) mm, rotated rx 37.25 ry 0 rz 3.74 deg; joints [122.723, -6.31, 56.765, -140.197, 57.613, 273.7, 25, -3.737]
  MoveL 977 to (-3.46, 91.17, -120.34) mm, rotated rx 37.25 ry 0 rz 3.74 deg; joints [122.713, -6.399, 56.789, -140.181, 57.559, 273.657, 25, -3.737]
  MoveL 978 to (-3.45, 91.36, -120.21) mm, rotated rx 37.33 ry 0 rz 3.72 deg; joints [122.695, -6.457, 56.793, -140.179, 57.51, 273.539, 25, -3.723]
  MoveL 979 to (-3.51, 91.87, -119.81) mm, rotated rx 37.33 ry 0 rz 3.72 deg; joints [122.683, -6.492, 56.795, -140.178, 57.48, 273.521, 25, -3.723]
  MoveL 980 to (-4.01, 93.64, -118.41) mm, rotated rx 38.19 ry 0 rz 3.96 deg; joints [122.509, -7.069, 56.838, -140.146, 56.998, 272.359, 25, -3.959]
  MoveL 981 to (-4, 93.62, -118.43) mm, rotated rx 38.58 ry 0 rz 3.93 deg; joints [122.448, -7.268, 56.849, -140.134, 56.829, 271.867, 25, -3.929]
  MoveL 982 to (-3.66, 94.95, -117.38) mm, rotated rx 39.22 ry 0 rz 3.67 deg; joints [122.322, -7.695, 56.873, -140.101, 56.467, 270.992, 25, -3.668]
  Set speed (16.7 mm/s)
  MoveL 983 to (-4.47, 107.57, -132.88) mm, rotated rx 39.22 ry 0 rz 3.67 deg; joints [121.667, -7.78, 57.365, -140.988, 56.51, 271.697, 25, -3.668]
  Set speed (1000.0 mm/s)
  MoveL 984 to (-3.83, 110.44, -130.52) mm, rotated rx 40.44 ry 0 rz 3.25 deg; joints [121.424, -8.62, 57.4, -140.914, 55.784, 270.015, 25, -3.247]
  Set speed (5.0 mm/s)
  MoveL 985 to (-3.09, 97.49, -115.3) mm, rotated rx 40.44 ry 0 rz 3.25 deg; joints [122.089, -8.504, 56.906, -140.021, 55.773, 269.314, 25, -3.247]
  Set speed (16.7 mm/s)
  MoveL 986 to (-2.24, 100.79, -112.45) mm, rotated rx 42.09 ry 0 rz 2.65 deg; joints [121.788, -9.579, 56.921, -139.879, 54.832, 267.017, 25, -2.653]
  MoveL 987 to (-2.17, 101.07, -112.19) mm, rotated rx 42.21 ry 0 rz 2.61 deg; joints [121.766, -9.661, 56.921, -139.866, 54.759, 266.844, 25, -2.613]
  MoveL 988 to (-1.61, 103.2, -110.24) mm, rotated rx 43.32 ry 0 rz 2.25 deg; joints [121.577, -10.364, 56.912, -139.746, 54.132, 265.298, 25, -2.247]
  MoveL 989 to (-1.56, 103.61, -109.86) mm, rotated rx 43.32 ry 0 rz 2.25 deg; joints [121.57, -10.395, 56.913, -139.739, 54.106, 265.279, 25, -2.247]
  MoveL 990 to (-1.57, 103.74, -109.74) mm, rotated rx 43.39 ry 0 rz 2.25 deg; joints [121.559, -10.44, 56.912, -139.731, 54.066, 265.179, 25, -2.247]
  MoveL 991 to (-1.73, 104.85, -108.68) mm, rotated rx 44.18 ry 0 rz 2.28 deg; joints [121.435, -10.906, 56.895, -139.64, 53.642, 264.084, 25, -2.277]
  MoveL 992 to (0.21, 108.08, -105.48) mm, rotated rx 46.08 ry 0 rz 1.09 deg; joints [121.139, -12.052, 56.821, -139.373, 52.579, 261.381, 25, -1.094]
  MoveL 993 to (0.42, 108.82, -104.72) mm, rotated rx 46.08 ry 0 rz 1.09 deg; joints [121.132, -12.115, 56.825, -139.353, 52.531, 261.338, 25, -1.094]
  MoveL 994 to (0.42, 109, -104.52) mm, rotated rx 46.19 ry 0 rz 1.1 deg; joints [121.117, -12.177, 56.82, -139.336, 52.473, 261.191, 25, -1.096]
  MoveL 995 to (0.32, 109.44, -104.07) mm, rotated rx 46.19 ry 0 rz 1.1 deg; joints [121.107, -12.204, 56.814, -139.33, 52.444, 261.171, 25, -1.096]
  MoveL 996 to (-0.31, 110.94, -102.46) mm, rotated rx 47.02 ry 0 rz 1.41 deg; joints [120.987, -12.705, 56.768, -139.188, 51.974, 259.969, 25, -1.405]
  MoveL 997 to (-0.3, 112.04, -101.27) mm, rotated rx 47.89 ry 0 rz 1.43 deg; joints [120.875, -13.194, 56.718, -139.035, 51.513, 258.723, 25, -1.433]
  MoveL 998 to (-0.34, 112.34, -100.94) mm, rotated rx 47.89 ry 0 rz 1.43 deg; joints [120.869, -13.214, 56.714, -139.03, 51.493, 258.707, 25, -1.433]
  MoveL 999 to (-0.39, 112.51, -100.74) mm, rotated rx 48 ry 0 rz 1.46 deg; joints [120.856, -13.273, 56.707, -139.01, 51.437, 258.56, 25, -1.456]
  MoveL 1000 to (-0.45, 112.67, -100.56) mm, rotated rx 48 ry 0 rz 1.46 deg; joints [120.852, -13.282, 56.704, -139.008, 51.426, 258.553, 25, -1.456]
  MoveL 1001 to (-1.06, 113.99, -99.05) mm, rotated rx 49.06 ry 0 rz 1.79 deg; joints [120.723, -13.868, 56.629, -138.804, 50.866, 257.018, 25, -1.789]
  MoveL 1002 to (-0.89, 116.98, -95.51) mm, rotated rx 51.11 ry 0 rz 1.57 deg; joints [120.481, -14.977, 56.435, -138.362, 49.769, 254.023, 25, -1.574]
  MoveL 1003 to (0.74, 119.64, -92.16) mm, rotated rx 52.74 ry 0 rz 0.76 deg; joints [120.309, -15.854, 56.247, -137.947, 48.889, 251.588, 25, -0.756]
  MoveL 1004 to (0.91, 120.12, -91.53) mm, rotated rx 52.74 ry 0 rz 0.76 deg; joints [120.306, -15.897, 56.245, -137.924, 48.855, 251.55, 25, -0.756]
  MoveL 1005 to (0.92, 120.24, -91.37) mm, rotated rx 52.82 ry 0 rz 0.75 deg; joints [120.299, -15.938, 56.235, -137.903, 48.813, 251.433, 25, -0.751]
  MoveL 1006 to (0.92, 120.42, -91.13) mm, rotated rx 52.82 ry 0 rz 0.75 deg; joints [120.296, -15.95, 56.232, -137.897, 48.8, 251.421, 25, -0.751]
  MoveL 1007 to (0.75, 121.59, -89.57) mm, rotated rx 53.74 ry 0 rz 0.82 deg; joints [120.212, -16.412, 56.114, -137.65, 48.327, 250.037, 25, -0.816]
  MoveL 1008 to (1.24, 122.75, -87.97) mm, rotated rx 54.6 ry 0 rz 0.55 deg; joints [120.137, -16.836, 55.994, -137.406, 47.887, 248.742, 25, -0.554]
  MoveL 1009 to (1.31, 123.04, -87.57) mm, rotated rx 54.6 ry 0 rz 0.55 deg; joints [120.135, -16.859, 55.991, -137.392, 47.867, 248.719, 25, -0.554]
  MoveL 1010 to (1.32, 123.17, -87.37) mm, rotated rx 54.69 ry 0 rz 0.55 deg; joints [120.127, -16.905, 55.978, -137.365, 47.819, 248.581, 25, -0.548]
  MoveL 1011 to (1.3, 123.44, -87) mm, rotated rx 54.69 ry 0 rz 0.55 deg; joints [120.124, -16.922, 55.972, -137.354, 47.8, 248.562, 25, -0.548]
  MoveL 1012 to (1, 124.63, -85.29) mm, rotated rx 55.56 ry 0 rz 0.69 deg; joints [120.056, -17.345, 55.842, -137.09, 47.359, 247.239, 25, -0.689]
  MoveL 1013 to (0.97, 124.77, -85.09) mm, rotated rx 55.76 ry 0 rz 0.7 deg; joints [120.042, -17.432, 55.814, -137.033, 47.267, 246.94, 25, -0.702]
  MoveL 1014 to (1.26, 127.48, -80.96) mm, rotated rx 57.64 ry 0 rz 0.55 deg; joints [119.915, -18.319, 55.496, -136.404, 46.321, 244.032, 25, -0.554]
  MoveL 1015 to (1.26, 127.68, -80.64) mm, rotated rx 57.64 ry 0 rz 0.55 deg; joints [119.913, -18.333, 55.49, -136.393, 46.306, 244.015, 25, -0.554]
  MoveL 1016 to (1.24, 127.76, -80.51) mm, rotated rx 57.7 ry 0 rz 0.56 deg; joints [119.91, -18.359, 55.48, -136.373, 46.277, 243.926, 25, -0.56]
  MoveL 1017 to (1.19, 127.95, -80.22) mm, rotated rx 57.7 ry 0 rz 0.56 deg; joints [119.907, -18.37, 55.473, -136.365, 46.263, 243.912, 25, -0.56]
  MoveL 1018 to (0.96, 128.4, -79.5) mm, rotated rx 58.28 ry 0 rz 0.68 deg; joints [119.878, -18.611, 55.379, -136.175, 46.005, 243.034, 25, -0.684]
  MoveL 1019 to (0.97, 128.48, -79.36) mm, rotated rx 58.34 ry 0 rz 0.68 deg; joints [119.875, -18.638, 55.368, -136.153, 45.976, 242.94, 25, -0.681]
  MoveL 1020 to (1.52, 130.36, -76.23) mm, rotated rx 59.82 ry 0 rz 0.42 deg; joints [119.803, -19.278, 55.081, -135.605, 45.27, 240.61, 25, -0.417]
  MoveL 1021 to (1.55, 130.51, -75.97) mm, rotated rx 59.82 ry 0 rz 0.42 deg; joints [119.802, -19.291, 55.077, -135.595, 45.258, 240.594, 25, -0.417]
  MoveL 1022 to (1.57, 130.9, -75.29) mm, rotated rx 60.12 ry 0 rz 0.41 deg; joints [119.79, -19.416, 55.017, -135.48, 45.119, 240.126, 25, -0.408]
  MoveL 1023 to (1.66, 133.76, -70.09) mm, rotated rx 62.52 ry 0 rz 0.34 deg; joints [119.717, -20.374, 54.499, -134.505, 44.032, 236.291, 25, -0.342]
  MoveL 1024 to (1.75, 133.98, -69.66) mm, rotated rx 62.71 ry 0 rz 0.3 deg; joints [119.713, -20.444, 54.457, -134.426, 43.951, 235.997, 25, -0.302]
  MoveL 1025 to (2.41, 135.04, -67.57) mm, rotated rx 63.67 ry 0 rz 0 deg; joints [119.698, -20.8, 54.23, -134.009, 43.536, 234.439, 25, 0]
  MoveL 1026 to (3, 135.96, -65.67) mm, rotated rx 64.48 ry 0 rz -0.25 deg; joints [119.691, -21.091, 54.034, -133.643, 43.195, 233.126, 25, 0.251]
  MoveL 1027 to (2.98, 135.95, -65.68) mm, rotated rx 65 ry 0 rz -0.66 deg; joints [119.668, -21.185, 53.898, -133.492, 43.023, 232.385, 25, 0.655]
  MoveL 1028 to (7.92, 137.22, -62.57) mm, rotated rx 66.39 ry 0 rz -2.88 deg; joints [119.665, -21.629, 53.528, -132.853, 42.463, 230.117, 25, 2.885]
  MoveL 1029 to (8.14, 137.25, -62.48) mm, rotated rx 66.43 ry 0 rz -2.98 deg; joints [119.665, -21.642, 53.518, -132.835, 42.448, 230.056, 25, 2.976]
  MoveL 1030 to (11.32, 137.44, -61.55) mm, rotated rx 66.85 ry 0 rz -4.39 deg; joints [119.665, -21.764, 53.4, -132.641, 42.285, 229.373, 25, 4.389]
  MoveL 1031 to (11.54, 137.46, -61.48) mm, rotated rx 66.85 ry 0 rz -4.39 deg; joints [119.67, -21.777, 53.405, -132.63, 42.283, 229.361, 25, 4.389]
  MoveL 1032 to (12.41, 137.53, -61.14) mm, rotated rx 66.99 ry 0 rz -4.75 deg; joints [119.672, -21.822, 53.367, -132.56, 42.228, 229.127, 25, 4.748]
  MoveL 1033 to (12.81, 137.58, -60.95) mm, rotated rx 66.99 ry 0 rz -4.75 deg; joints [119.681, -21.847, 53.376, -132.536, 42.222, 229.102, 25, 4.748]
  MoveL 1034 to (16.95, 138.2, -58.48) mm, rotated rx 68.01 ry 0 rz -6.43 deg; joints [119.701, -22.164, 53.096, -132.024, 41.833, 227.405, 25, 6.43]
  MoveL 1035 to (21.14, 138.65, -56) mm, rotated rx 69.03 ry 0 rz -8.11 deg; joints [119.728, -22.464, 52.807, -131.497, 41.458, 225.699, 25, 8.113]
  MoveL 1036 to (22.1, 138.9, -55.01) mm, rotated rx 69.03 ry 0 rz -8.11 deg; joints [119.751, -22.535, 52.813, -131.416, 41.43, 225.606, 25, 8.113]
  MoveL 1037 to (22.2, 138.96, -54.82) mm, rotated rx 69.11 ry 0 rz -8.15 deg; joints [119.753, -22.557, 52.791, -131.376, 41.402, 225.477, 25, 8.151]
  MoveL 1038 to (22.35, 139.07, -54.48) mm, rotated rx 69.11 ry 0 rz -8.15 deg; joints [119.757, -22.572, 52.787, -131.355, 41.392, 225.452, 25, 8.151]
  MoveL 1039 to (22.88, 139.59, -52.91) mm, rotated rx 69.96 ry 0 rz -8.43 deg; joints [119.782, -22.784, 52.543, -130.936, 41.109, 224.062, 25, 8.429]
  MoveL 1040 to (25.99, 140.24, -49.64) mm, rotated rx 71.43 ry 0 rz -9.74 deg; joints [119.841, -23.144, 52.099, -130.161, 40.625, 221.603, 25, 9.739]
  MoveL 1041 to (26.74, 140.41, -48.75) mm, rotated rx 71.74 ry 0 rz -9.99 deg; joints [119.86, -23.228, 52.003, -129.979, 40.523, 221.068, 25, 9.986]
  MoveL 1042 to (32.5, 141.63, -41.13) mm, rotated rx 74.73 ry 0 rz -12.11 deg; joints [120.061, -23.895, 51.039, -128.248, 39.631, 215.936, 25, 12.11]
  MoveL 1043 to (32.75, 141.66, -40.84) mm, rotated rx 74.89 ry 0 rz -12.24 deg; joints [120.071, -23.921, 50.986, -128.162, 39.589, 215.671, 25, 12.238]
  MoveL 1044 to (35.63, 141.87, -37.54) mm, rotated rx 76.2 ry 0 rz -13.34 deg; joints [120.181, -24.163, 50.54, -127.377, 39.245, 213.405, 25, 13.337]
  MoveL 1045 to (38.54, 141.6, -35.67) mm, rotated rx 77.13 ry 0 rz -14.68 deg; joints [120.251, -24.286, 50.217, -126.862, 39.026, 211.859, 25, 14.681]
  MoveL 1046 to (38.93, 141.57, -35.36) mm, rotated rx 77.13 ry 0 rz -14.68 deg; joints [120.262, -24.309, 50.22, -126.831, 39.022, 211.825, 25, 14.681]
  MoveL 1047 to (39.55, 141.62, -34.44) mm, rotated rx 77.13 ry 0 rz -14.68 deg; joints [120.282, -24.351, 50.213, -126.76, 39.008, 211.745, 25, 14.681]
  MoveL 1048 to (39.7, 141.67, -34.05) mm, rotated rx 77.28 ry 0 rz -14.74 deg; joints [120.297, -24.376, 50.159, -126.666, 38.972, 211.48, 25, 14.735]
  MoveL 1049 to (41.12, 142.09, -30.47) mm, rotated rx 78.67 ry 0 rz -15.22 deg; joints [120.442, -24.584, 49.664, -125.802, 38.661, 209.06, 25, 15.223]
  MoveL 1050 to (41.26, 142.16, -29.95) mm, rotated rx 78.67 ry 0 rz -15.22 deg; joints [120.45, -24.596, 49.652, -125.77, 38.653, 209.023, 25, 15.223]
  MoveL 1051 to (41.16, 142.43, -28.75) mm, rotated rx 78.67 ry 0 rz -15.22 deg; joints [120.457, -24.601, 49.612, -125.716, 38.631, 208.957, 25, 15.223]
  MoveL 1052 to (41.03, 142.55, -28.37) mm, rotated rx 78.82 ry 0 rz -15.16 deg; joints [120.473, -24.622, 49.557, -125.621, 38.6, 208.696, 25, 15.161]
  MoveL 1053 to (40.52, 142.86, -27.52) mm, rotated rx 78.82 ry 0 rz -15.16 deg; joints [120.468, -24.602, 49.513, -125.602, 38.582, 208.668, 25, 15.161]
  MoveL 1054 to (38.89, 143.61, -25.84) mm, rotated rx 79.47 ry 0 rz -14.48 deg; joints [120.543, -24.686, 49.277, -125.194, 38.451, 207.538, 25, 14.483]
  MoveL 1055 to (38.92, 143.6, -25.89) mm, rotated rx 80.77 ry 0 rz -14.46 deg; joints [120.669, -24.811, 48.901, -124.539, 38.259, 205.463, 25, 14.458]
  MoveL 1056 to (39.51, 143.55, -25.27) mm, rotated rx 81.01 ry 0 rz -14.68 deg; joints [120.698, -24.837, 48.812, -124.387, 38.216, 205.047, 25, 14.681]
  MoveL 1057 to (40.07, 143.56, -24.36) mm, rotated rx 81.01 ry 0 rz -14.68 deg; joints [120.72, -24.872, 48.802, -124.317, 38.207, 204.969, 25, 14.681]
  MoveL 1058 to (40.29, 143.6, -23.74) mm, rotated rx 81.25 ry 0 rz -14.76 deg; joints [120.75, -24.897, 48.713, -124.166, 38.166, 204.558, 25, 14.758]
  MoveL 1059 to (40.41, 143.65, -23.24) mm, rotated rx 81.25 ry 0 rz -14.76 deg; joints [120.758, -24.906, 48.701, -124.135, 38.16, 204.523, 25, 14.758]
  MoveL 1060 to (40.3, 143.86, -22.08) mm, rotated rx 81.25 ry 0 rz -14.76 deg; joints [120.767, -24.908, 48.661, -124.081, 38.143, 204.459, 25, 14.758]
  MoveL 1061 to (38.72, 144.91, -17.54) mm, rotated rx 82.98 ry 0 rz -14.07 deg; joints [121.003, -25.062, 47.997, -122.962, 37.872, 201.421, 25, 14.072]
  MoveL 1062 to (38.58, 144.99, -17.22) mm, rotated rx 82.98 ry 0 rz -14.07 deg; joints [121.003, -25.057, 47.982, -122.951, 37.867, 201.407, 25, 14.072]
  MoveL 1063 to (38.48, 145.04, -17.03) mm, rotated rx 83.05 ry 0 rz -14.03 deg; joints [121.013, -25.062, 47.955, -122.906, 37.857, 201.284, 25, 14.032]
  MoveL 1064 to (37.63, 145.45, -15.32) mm, rotated rx 83.73 ry 0 rz -13.67 deg; joints [121.112, -25.111, 47.695, -122.47, 37.767, 200.106, 25, 13.665]
  MoveL 1065 to (37.23, 145.61, -14.75) mm, rotated rx 83.73 ry 0 rz -13.67 deg; joints [121.109, -25.093, 47.664, -122.458, 37.757, 200.09, 25, 13.665]
  MoveL 1066 to (37.03, 145.69, -14.54) mm, rotated rx 83.81 ry 0 rz -13.58 deg; joints [121.121, -25.099, 47.632, -122.404, 37.747, 199.946, 25, 13.584]
  MoveL 1067 to (36.58, 145.84, -14.17) mm, rotated rx 83.81 ry 0 rz -13.58 deg; joints [121.115, -25.078, 47.605, -122.404, 37.739, 199.943, 25, 13.584]
  MoveL 1068 to (34.46, 146.47, -12.81) mm, rotated rx 84.32 ry 0 rz -12.74 deg; joints [121.193, -25.109, 47.402, -122.069, 37.675, 199.041, 25, 12.739]
  MoveL 1069 to (34.47, 146.47, -12.84) mm, rotated rx 84.6 ry 0 rz -12.45 deg; joints [121.244, -25.159, 47.342, -121.896, 37.656, 198.57, 25, 12.448]
  MoveL 1070 to (33.46, 146.84, -11.22) mm, rotated rx 85.22 ry 0 rz -12.04 deg; joints [121.34, -25.19, 47.097, -121.494, 37.587, 197.492, 25, 12.041]
  MoveL 1071 to (33.09, 146.96, -10.77) mm, rotated rx 85.22 ry 0 rz -12.04 deg; joints [121.337, -25.174, 47.07, -121.486, 37.58, 197.48, 25, 12.041]
  MoveL 1072 to (32.68, 147.08, -10.37) mm, rotated rx 85.37 ry 0 rz -11.88 deg; joints [121.361, -25.18, 47.01, -121.387, 37.564, 197.215, 25, 11.878]
  MoveL 1073 to (32.51, 147.13, -10.22) mm, rotated rx 85.37 ry 0 rz -11.88 deg; joints [121.359, -25.172, 46.999, -121.387, 37.561, 197.213, 25, 11.878]
  MoveL 1074 to (29.75, 147.84, -8.03) mm, rotated rx 86.2 ry 0 rz -10.8 deg; joints [121.495, -25.204, 46.665, -120.845, 37.48, 195.761, 25, 10.797]
  MoveL 1075 to (29.76, 147.84, -8.04) mm, rotated rx 86.94 ry 0 rz -10.43 deg; joints [121.614, -25.267, 46.46, -120.425, 37.439, 194.546, 25, 10.432]
  MoveL 1076 to (29.76, 148.04, -2.01) mm, rotated rx 89.23 ry 0 rz -10.42 deg; joints [122.02, -25.291, 45.518, -118.937, 37.291, 190.567, 25, 10.418]
  MoveL 1077 to (29.74, 148.04, -2.09) mm, rotated rx 89.77 ry 0 rz -10.59 deg; joints [122.087, -25.265, 45.329, -118.687, 37.266, 189.742, 25, 10.592]
  MoveL 1078 to (31.21, 147.76, -0.05) mm, rotated rx 90.54 ry 0 rz -11.16 deg; joints [122.233, -25.255, 45.004, -118.187, 37.238, 188.404, 25, 11.161]
  MoveL 1079 to (31.48, 147.7, 0.47) mm, rotated rx 90.85 ry 0 rz -11.36 deg; joints [122.283, -25.237, 44.877, -118.014, 37.227, 187.9, 25, 11.36]
  MoveL 1080 to (32.83, 147.39, 1.86) mm, rotated rx 91.38 ry 0 rz -11.88 deg; joints [122.386, -25.224, 44.654, -117.676, 37.216, 186.993, 25, 11.884]
  MoveL 1081 to (32.8, 147.39, 1.84) mm, rotated rx 91.48 ry 0 rz -13.08 deg; joints [122.329, -25.073, 44.523, -117.75, 37.177, 186.956, 25, 13.082]
  MoveL 1082 to (33.53, 147.24, 1.33) mm, rotated rx 91.29 ry 0 rz -13.37 deg; joints [122.291, -25.079, 44.605, -117.874, 37.181, 187.29, 25, 13.365]
  MoveL 1083 to (33.53, 147.25, 1.3) mm, rotated rx 91.01 ry 0 rz -13.62 deg; joints [122.233, -25.053, 44.677, -118.041, 37.179, 187.749, 25, 13.62]
  MoveL 1084 to (34.87, 146.94, -0.79) mm, rotated rx 90.22 ry 0 rz -14.14 deg; joints [122.081, -25.068, 45.01, -118.551, 37.203, 189.115, 25, 14.141]
  MoveL 1085 to (35.62, 146.75, -1.54) mm, rotated rx 90.22 ry 0 rz -14.14 deg; joints [122.087, -25.105, 45.059, -118.56, 37.214, 189.128, 25, 14.141]
  MoveL 1086 to (36.61, 146.5, -1.89) mm, rotated rx 90.22 ry 0 rz -14.14 deg; joints [122.104, -25.153, 45.102, -118.537, 37.226, 189.108, 25, 14.141]
  MoveL 1087 to (37.17, 146.36, -1.96) mm, rotated rx 90.2 ry 0 rz -14.36 deg; joints [122.1, -25.153, 45.113, -118.554, 37.227, 189.152, 25, 14.359]
  MoveL 1088 to (37.6, 146.25, -1.97) mm, rotated rx 90.2 ry 0 rz -14.36 deg; joints [122.109, -25.174, 45.127, -118.537, 37.232, 189.135, 25, 14.359]
  MoveL 1089 to (38.54, 146.01, -1.71) mm, rotated rx 90.2 ry 0 rz -14.36 deg; joints [122.135, -25.219, 45.148, -118.484, 37.242, 189.08, 25, 14.359]
  MoveL 1090 to (42.69, 144.86, 0.45) mm, rotated rx 91.02 ry 0 rz -15.99 deg; joints [122.294, -25.204, 44.801, -117.955, 37.217, 187.66, 25, 15.994]
  MoveL 1091 to (45.11, 144.13, 0.77) mm, rotated rx 91.23 ry 0 rz -17.25 deg; joints [122.313, -25.162, 44.695, -117.861, 37.203, 187.336, 25, 17.255]
  Set speed (16.7 mm/s)
  MoveL 1092 to (59.93, 191.86, 1.85) mm, rotated rx 91.23 ry 0 rz -17.25 deg; joints [120.667, -26.712, 44.887, -117.744, 35.191, 186.532, 25, 17.255]
  Set speed (5.0 mm/s)
  Call SetCLW
  Call SetRPM(70.0)
  MoveL 1093 to (-167.66, 48.48, 99.74) mm, rotated rx 119.08 ry 0 rz 74.16 deg; joints [128.785, -21.422, 31.151, -101.876, 39.799, 141.227, 25, -74.158]
  MoveL 1094 to (-125.62, 36.55, 75.44) mm, rotated rx 119.08 ry 0 rz 74.16 deg; joints [129.673, -20.393, 31.864, -103.483, 41.034, 143.553, 25, -74.158]
  Set speed (16.7 mm/s)
  MoveL 1095 to (-125.66, 36.09, 75.59) mm, rotated rx 119.15 ry 0 rz 74.36 deg; joints [129.693, -20.374, 31.834, -103.461, 41.05, 143.464, 25, -74.359]
  MoveL 1096 to (-126.55, 30.63, 76.51) mm, rotated rx 119.51 ry 0 rz 76.59 deg; joints [129.794, -20.251, 31.649, -103.346, 41.132, 142.977, 25, -76.593]
  MoveL 1097 to (-126.75, 29.66, 76.56) mm, rotated rx 119.51 ry 0 rz 76.87 deg; joints [129.788, -20.234, 31.634, -103.351, 41.127, 142.974, 25, -76.868]
  MoveL 1098 to (-128.06, 23.4, 76.55) mm, rotated rx 119.51 ry 0 rz 79.64 deg; joints [129.784, -20.233, 31.635, -103.356, 41.123, 142.987, 25, -79.642]
  MoveL 1099 to (-128.14, 21.08, 77.09) mm, rotated rx 119.77 ry 0 rz 80.93 deg; joints [129.877, -20.18, 31.53, -103.255, 41.201, 142.612, 25, -80.928]
  MoveL 1100 to (-128.27, 20.02, 77.16) mm, rotated rx 119.78 ry 0 rz 81.16 deg; joints [129.867, -20.156, 31.51, -103.264, 41.192, 142.616, 25, -81.155]
  MoveL 1101 to (-129.21, 15.23, 76.67) mm, rotated rx 119.57 ry 0 rz 83.14 deg; joints [129.795, -20.204, 31.599, -103.343, 41.132, 142.91, 25, -83.143]
  MoveL 1102 to (-129.09, 12.94, 77.31) mm, rotated rx 119.88 ry 0 rz 84.58 deg; joints [129.911, -20.153, 31.484, -103.219, 41.228, 142.466, 25, -84.585]
  MoveL 1103 to (-129.13, 12.06, 77.39) mm, rotated rx 119.88 ry 0 rz 84.58 deg; joints [129.891, -20.117, 31.457, -103.237, 41.211, 142.484, 25, -84.585]
  MoveL 1104 to (-129.47, 10.56, 77.03) mm, rotated rx 119.87 ry 0 rz 84.75 deg; joints [129.851, -20.086, 31.445, -103.276, 41.177, 142.537, 25, -84.749]
  MoveL 1105 to (-130.4, 8.24, 75.73) mm, rotated rx 119.29 ry 0 rz 85.8 deg; joints [129.677, -20.254, 31.713, -103.468, 41.035, 143.322, 25, -85.803]
  MoveL 1106 to (-131.29, 7.17, 74.28) mm, rotated rx 119.29 ry 0 rz 85.8 deg; joints [129.609, -20.25, 31.745, -103.54, 40.978, 143.399, 25, -85.803]
  MoveL 1107 to (-131.73, 7.15, 73.51) mm, rotated rx 119.24 ry 0 rz 85.81 deg; joints [129.575, -20.28, 31.796, -103.578, 40.951, 143.49, 25, -85.813]
  MoveL 1108 to (-132.2, 7.3, 72.65) mm, rotated rx 118.87 ry 0 rz 85.76 deg; joints [129.463, -20.388, 31.971, -103.707, 40.86, 144.005, 25, -85.763]
  MoveL 1109 to (-132.78, 6.62, 71.65) mm, rotated rx 117.86 ry 0 rz 86.21 deg; joints [129.204, -20.65, 32.394, -104.011, 40.652, 145.351, 25, -86.21]
  MoveL 1110 to (-133.74, 6.48, 69.85) mm, rotated rx 117.86 ry 0 rz 86.21 deg; joints [129.151, -20.688, 32.465, -104.074, 40.609, 145.42, 25, -86.21]
  MoveL 1111 to (-134.44, 7.5, 68.38) mm, rotated rx 116.1 ry 0 rz 86.27 deg; joints [128.728, -21.142, 33.203, -104.604, 40.279, 147.752, 25, -86.267]
  MoveL 1112 to (-134.6, 7.01, 68.11) mm, rotated rx 115.99 ry 0 rz 86.48 deg; joints [128.694, -21.172, 33.255, -104.646, 40.253, 147.91, 25, -86.48]
  MoveL 1113 to (-135.14, 4.27, 67.26) mm, rotated rx 115.55 ry 0 rz 87.85 deg; joints [128.58, -21.302, 33.466, -104.796, 40.166, 148.516, 25, -87.845]
  MoveL 1114 to (-135.12, 2.4, 67.41) mm, rotated rx 115.57 ry 0 rz 89.05 deg; joints [128.612, -21.334, 33.481, -104.761, 40.191, 148.465, 25, -89.054]
  MoveL 1115 to (-135.16, 1.48, 67.35) mm, rotated rx 115.54 ry 0 rz 89.24 deg; joints [128.593, -21.321, 33.478, -104.782, 40.176, 148.509, 25, -89.239]
  MoveL 1116 to (-135.48, -0.78, 66.72) mm, rotated rx 115.35 ry 0 rz 90 deg; joints [128.521, -21.357, 33.562, -104.874, 40.12, 148.798, 25, -90]
  MoveL 1117 to (-135.78, -3.03, 66.05) mm, rotated rx 115.03 ry 0 rz 90.95 deg; joints [128.428, -21.438, 33.708, -104.995, 40.049, 149.253, 25, -90.95]
  MoveL 1118 to (-135.91, -3.72, 65.73) mm, rotated rx 115.03 ry 0 rz 90.95 deg; joints [128.404, -21.419, 33.703, -105.024, 40.029, 149.283, 25, -90.95]
  MoveL 1119 to (-136.03, -4.12, 65.47) mm, rotated rx 114.92 ry 0 rz 91.12 deg; joints [128.371, -21.448, 33.755, -105.067, 40.005, 149.442, 25, -91.121]
  MoveL 1120 to (-136.91, -6.5, 63.38) mm, rotated rx 114.14 ry 0 rz 91.98 deg; joints [128.13, -21.639, 34.119, -105.392, 39.823, 150.575, 25, -91.982]
  MoveL 1121 to (-136.91, -6.56, 63.38) mm, rotated rx 113.87 ry 0 rz 92.66 deg; joints [128.105, -21.755, 34.263, -105.438, 39.807, 150.902, 25, -92.66]
  MoveL 1122 to (-136.87, -8.62, 63.24) mm, rotated rx 113.81 ry 0 rz 93.52 deg; joints [128.086, -21.771, 34.292, -105.463, 39.793, 150.992, 25, -93.521]
  MoveL 1123 to (-136.9, -9.7, 63.03) mm, rotated rx 113.75 ry 0 rz 93.81 deg; joints [128.057, -21.773, 34.314, -105.501, 39.771, 151.096, 25, -93.811]
  MoveL 1124 to (-137.08, -13.18, 61.94) mm, rotated rx 113.32 ry 0 rz 95.15 deg; joints [127.926, -21.87, 34.509, -105.685, 39.674, 151.724, 25, -95.153]
  MoveL 1125 to (-137.06, -13.23, 61.99) mm, rotated rx 113.99 ry 0 rz 96.52 deg; joints [128.159, -21.866, 34.351, -105.383, 39.852, 150.73, 25, -96.517]
  MoveL 1126 to (-136.35, -13.61, 63.48) mm, rotated rx 114.61 ry 0 rz 96.71 deg; joints [128.341, -21.709, 34.06, -105.134, 39.988, 149.836, 25, -96.706]
  MoveL 1127 to (-135.76, -14.07, 64.65) mm, rotated rx 114.97 ry 0 rz 96.88 deg; joints [128.453, -21.603, 33.874, -104.983, 40.073, 149.304, 25, -96.878]
  MoveL 1128 to (-135.39, -14.51, 65.31) mm, rotated rx 114.97 ry 0 rz 96.88 deg; joints [128.459, -21.569, 33.833, -104.973, 40.077, 149.292, 25, -96.878]
  MoveL 1129 to (-134.85, -16.26, 66.02) mm, rotated rx 114.97 ry 0 rz 96.88 deg; joints [128.433, -21.482, 33.754, -104.995, 40.054, 149.313, 25, -96.878]
  MoveL 1130 to (-133.31, -26, 66.04) mm, rotated rx 114.98 ry 0 rz 101.04 deg; joints [128.435, -21.48, 33.75, -104.991, 40.056, 149.301, 25, -101.038]
  MoveL 1131 to (-133.19, -26.82, 65.93) mm, rotated rx 114.96 ry 0 rz 101.19 deg; joints [128.415, -21.469, 33.75, -105.015, 40.039, 149.353, 25, -101.185]
  MoveL 1132 to (-132.71, -29.77, 65.64) mm, rotated rx 114.82 ry 0 rz 102.53 deg; joints [128.381, -21.511, 33.817, -105.062, 40.014, 149.539, 25, -102.527]
  MoveL 1133 to (-132.63, -30.55, 65.46) mm, rotated rx 114.79 ry 0 rz 102.62 deg; joints [128.355, -21.499, 33.821, -105.092, 39.994, 149.602, 25, -102.622]
  MoveL 1134 to (-132.62, -32.3, 64.62) mm, rotated rx 114.39 ry 0 rz 103.7 deg; joints [128.262, -21.634, 34.028, -105.225, 39.925, 150.152, 25, -103.703]
  MoveL 1135 to (-132.27, -33.65, 64.64) mm, rotated rx 114.39 ry 0 rz 104.29 deg; joints [128.264, -21.632, 34.025, -105.221, 39.926, 150.14, 25, -104.29]
  MoveL 1136 to (-132.01, -34.95, 64.49) mm, rotated rx 114.34 ry 0 rz 104.68 deg; joints [128.238, -21.63, 34.039, -105.254, 39.906, 150.228, 25, -104.676]
  MoveL 1137 to (-130.71, -42.04, 62.89) mm, rotated rx 113.68 ry 0 rz 108.03 deg; joints [128.064, -21.831, 34.374, -105.5, 39.777, 151.165, 25, -108.028]
  MoveL 1138 to (-128.93, -45.38, 64.23) mm, rotated rx 114.29 ry 0 rz 109.77 deg; joints [128.25, -21.697, 34.105, -105.246, 39.917, 150.276, 25, -109.774]
  MoveL 1139 to (-128.54, -46.25, 64.39) mm, rotated rx 114.29 ry 0 rz 109.77 deg; joints [128.231, -21.656, 34.072, -105.266, 39.901, 150.295, 25, -109.774]
  MoveL 1140 to (-128.24, -47.09, 64.38) mm, rotated rx 114.28 ry 0 rz 110.15 deg; joints [128.229, -21.657, 34.075, -105.268, 39.9, 150.303, 25, -110.147]
  MoveL 1141 to (-126.17, -53.24, 63.63) mm, rotated rx 113.98 ry 0 rz 112.74 deg; joints [128.134, -21.723, 34.209, -105.398, 39.828, 150.748, 25, -112.743]
  MoveL 1142 to (-126.2, -53.19, 63.61) mm, rotated rx 114.54 ry 0 rz 113.81 deg; joints [128.327, -21.714, 34.075, -105.153, 39.978, 149.921, 25, -113.815]
  MoveL 1143 to (-124.24, -53.95, 66.8) mm, rotated rx 115.89 ry 0 rz 114.45 deg; joints [128.723, -21.364, 33.448, -104.632, 40.28, 148.006, 25, -114.447]
  MoveL 1144 to (-123.99, -54.03, 67.19) mm, rotated rx 116.06 ry 0 rz 114.53 deg; joints [128.773, -21.319, 33.368, -104.568, 40.319, 147.764, 25, -114.526]
  MoveL 1145 to (-122.28, -54.76, 69.68) mm, rotated rx 117.48 ry 0 rz 115.19 deg; joints [129.177, -20.962, 32.746, -104.069, 40.636, 145.8, 25, -115.19]
  MoveL 1146 to (-121.62, -54.01, 71.37) mm, rotated rx 118.38 ry 0 rz 115.01 deg; joints [129.435, -20.717, 32.34, -103.764, 40.843, 144.562, 25, -115.006]
  Set speed (16.7 mm/s)
  MoveL 1147 to (-137.56, -61.45, 80.88) mm, rotated rx 118.38 ry 0 rz 115.01 deg; joints [129.074, -21.146, 32.071, -103.14, 40.336, 143.646, 25, -115.006]
  Set speed (1000.0 mm/s)
  MoveL 1148 to (-122.96, -67.13, 98.06) mm, rotated rx 125.73 ry 0 rz 119.11 deg; joints [131.309, -18.82, 28.59, -100.93, 42.246, 133.886, 25, -119.107]
  Set speed (5.0 mm/s)
  MoveL 1149 to (-108.78, -59.24, 86.38) mm, rotated rx 125.73 ry 0 rz 119.11 deg; joints [131.586, -18.465, 28.95, -101.589, 42.653, 134.845, 25, -119.107]
  Set speed (16.7 mm/s)
  MoveL 1150 to (-109.6, -55.06, 88.11) mm, rotated rx 126.53 ry 0 rz 117.22 deg; joints [131.83, -18.202, 28.581, -101.38, 42.867, 133.822, 25, -117.221]
  MoveL 1151 to (-109.69, -54.52, 88.34) mm, rotated rx 126.61 ry 0 rz 117.04 deg; joints [131.858, -18.18, 28.547, -101.357, 42.892, 133.723, 25, -117.04]
  MoveL 1152 to (-110.14, -49.87, 90.49) mm, rotated rx 127.62 ry 0 rz 114.99 deg; joints [132.167, -17.842, 28.082, -101.105, 43.165, 132.443, 25, -114.986]
  MoveL 1153 to (-110.47, -49.5, 90.29) mm, rotated rx 127.6 ry 0 rz 113.7 deg; joints [132.1, -17.774, 28.038, -101.156, 43.105, 132.516, 25, -113.701]
  MoveL 1154 to (-110.74, -49.15, 90.15) mm, rotated rx 127.54 ry 0 rz 113.5 deg; joints [132.08, -17.796, 28.068, -101.171, 43.087, 132.596, 25, -113.498]
  MoveL 1155 to (-113.2, -45.52, 89.01) mm, rotated rx 127.01 ry 0 rz 111.53 deg; joints [131.923, -17.977, 28.314, -101.3, 42.948, 133.256, 25, -111.533]
  MoveL 1156 to (-113.75, -44.17, 88.98) mm, rotated rx 127.01 ry 0 rz 111.53 deg; joints [131.958, -18.03, 28.354, -101.273, 42.98, 133.228, 25, -111.533]
  MoveL 1157 to (-113.85, -43.69, 89.08) mm, rotated rx 127.06 ry 0 rz 111.3 deg; joints [131.974, -18.013, 28.331, -101.26, 42.994, 133.164, 25, -111.302]
  MoveL 1158 to (-113.83, -42.24, 89.81) mm, rotated rx 127.06 ry 0 rz 111.3 deg; joints [132.03, -18.036, 28.333, -101.217, 43.044, 133.118, 25, -111.302]
  MoveL 1159 to (-112.96, -39.81, 91.98) mm, rotated rx 128.43 ry 0 rz 109.78 deg; joints [132.393, -17.555, 27.706, -100.927, 43.366, 131.446, 25, -109.783]
  MoveL 1160 to (-113.22, -37.92, 92.45) mm, rotated rx 128.65 ry 0 rz 108.89 deg; joints [132.462, -17.477, 27.602, -100.874, 43.428, 131.162, 25, -108.887]
  MoveL 1161 to (-113.16, -37.92, 92.52) mm, rotated rx 128.37 ry 0 rz 107.58 deg; joints [132.328, -17.453, 27.627, -100.974, 43.308, 131.549, 25, -107.58]
  MoveL 1162 to (-115.33, -36.4, 90.44) mm, rotated rx 127.39 ry 0 rz 106.59 deg; joints [132.027, -17.789, 28.081, -101.213, 43.04, 132.79, 25, -106.59]
  MoveL 1163 to (-116.24, -35.64, 89.58) mm, rotated rx 127.03 ry 0 rz 106.19 deg; joints [131.92, -17.915, 28.252, -101.301, 42.945, 133.234, 25, -106.189]
  MoveL 1164 to (-117, -35.63, 88.59) mm, rotated rx 126.27 ry 0 rz 105.85 deg; joints [131.693, -18.13, 28.561, -101.489, 42.746, 134.203, 25, -105.846]
  MoveL 1165 to (-117.3, -35.53, 88.23) mm, rotated rx 126.1 ry 0 rz 105.76 deg; joints [131.643, -18.185, 28.638, -101.533, 42.701, 134.416, 25, -105.765]
  MoveL 1166 to (-118.82, -34.81, 86.45) mm, rotated rx 125.36 ry 0 rz 105.3 deg; joints [131.414, -18.437, 28.992, -101.732, 42.502, 135.371, 25, -105.298]
  MoveL 1167 to (-119.06, -35.54, 85.84) mm, rotated rx 123.71 ry 0 rz 106.86 deg; joints [131.069, -18.973, 29.695, -102.051, 42.204, 137.365, 25, -106.862]
  MoveL 1168 to (-118.72, -36.4, 85.95) mm, rotated rx 123.74 ry 0 rz 107.02 deg; joints [131.065, -18.942, 29.664, -102.053, 42.201, 137.338, 25, -107.024]
  MoveL 1169 to (-117.63, -39.9, 85.89) mm, rotated rx 123.72 ry 0 rz 108.72 deg; joints [131.058, -18.95, 29.676, -102.061, 42.194, 137.371, 25, -108.717]
  MoveL 1170 to (-117.55, -40.02, 85.95) mm, rotated rx 123.86 ry 0 rz 109.35 deg; joints [131.124, -18.958, 29.655, -102.002, 42.252, 137.169, 25, -109.354]
  MoveL 1171 to (-116.07, -42, 87.01) mm, rotated rx 124.35 ry 0 rz 110.45 deg; joints [131.274, -18.8, 29.426, -101.865, 42.382, 136.526, 25, -110.449]
  MoveL 1172 to (-115.72, -42.53, 87.22) mm, rotated rx 124.38 ry 0 rz 110.56 deg; joints [131.278, -18.772, 29.395, -101.86, 42.385, 136.49, 25, -110.559]
  MoveL 1173 to (-114.38, -45.11, 87.69) mm, rotated rx 124.56 ry 0 rz 111.74 deg; joints [131.328, -18.698, 29.297, -101.815, 42.427, 136.258, 25, -111.737]
  MoveL 1174 to (-113.68, -46.83, 87.7) mm, rotated rx 124.55 ry 0 rz 112.36 deg; joints [131.312, -18.681, 29.287, -101.828, 42.414, 136.283, 25, -112.361]
  MoveL 1175 to (-110.62, -57.25, 85.4) mm, rotated rx 123.52 ry 0 rz 117.07 deg; joints [130.981, -18.993, 29.754, -102.131, 42.128, 137.644, 25, -117.068]
  MoveL 1176 to (-109.2, -59.64, 85.56) mm, rotated rx 123.57 ry 0 rz 118.71 deg; joints [131.017, -19.004, 29.751, -102.1, 42.159, 137.564, 25, -118.709]
  MoveL 1177 to (-109.19, -59.64, 85.56) mm, rotated rx 124.69 ry 0 rz 119.78 deg; joints [131.345, -18.804, 29.402, -101.805, 42.444, 136.121, 25, -119.778]
  MoveL 1178 to (-108.79, -59.2, 86.38) mm, rotated rx 125.07 ry 0 rz 119.69 deg; joints [131.46, -18.682, 29.227, -101.702, 42.544, 135.633, 25, -119.694]
  Set speed (16.7 mm/s)
  MoveL 1179 to (-123.01, -67.31, 97.87) mm, rotated rx 125.07 ry 0 rz 119.69 deg; joints [131.175, -19.044, 28.875, -101.046, 42.128, 134.677, 25, -119.694]
  Set speed (1000.0 mm/s)
  MoveL 1180 to (-103.64, -86, 105.37) mm, rotated rx 128.85 ry 0 rz 129.44 deg; joints [132.245, -17.684, 27.079, -100.19, 43.085, 129.972, 25, -129.439]
  Set speed (5.0 mm/s)
  MoveL 1181 to (-91.61, -76.1, 92.82) mm, rotated rx 128.85 ry 0 rz 129.44 deg; joints [132.488, -17.362, 27.476, -100.853, 43.451, 130.939, 25, -129.439]
  Set speed (16.7 mm/s)
  MoveL 1182 to (-93.41, -74.47, 92.39) mm, rotated rx 128.64 ry 0 rz 128.29 deg; joints [132.423, -17.436, 27.574, -100.902, 43.393, 131.205, 25, -128.287]
  MoveL 1183 to (-95.35, -73.29, 91.34) mm, rotated rx 128.03 ry 0 rz 126.93 deg; joints [132.225, -17.611, 27.825, -101.055, 43.216, 131.98, 25, -126.929]
  MoveL 1184 to (-95.55, -73.36, 91.06) mm, rotated rx 126.5 ry 0 rz 126.58 deg; joints [131.834, -18, 28.372, -101.372, 42.87, 133.845, 25, -126.585]
  MoveL 1185 to (-95.55, -74.38, 90.24) mm, rotated rx 126.11 ry 0 rz 126.97 deg; joints [131.715, -18.13, 28.553, -101.472, 42.765, 134.344, 25, -126.972]
  MoveL 1186 to (-95.64, -74.93, 89.7) mm, rotated rx 126.11 ry 0 rz 126.97 deg; joints [131.689, -18.135, 28.568, -101.493, 42.742, 134.367, 25, -126.972]
  MoveL 1187 to (-95.78, -75.25, 89.28) mm, rotated rx 126.04 ry 0 rz 127 deg; joints [131.657, -18.163, 28.609, -101.52, 42.714, 134.465, 25, -127.004]
  MoveL 1188 to (-96.18, -75.88, 88.31) mm, rotated rx 125.59 ry 0 rz 127.13 deg; joints [131.519, -18.311, 28.819, -101.639, 42.593, 135.046, 25, -127.129]
  MoveL 1189 to (-95.54, -78.96, 86.28) mm, rotated rx 124.14 ry 0 rz 128.8 deg; joints [131.13, -18.772, 29.46, -101.989, 42.255, 136.871, 25, -128.8]
  MoveL 1190 to (-95.44, -79.45, 85.95) mm, rotated rx 124.04 ry 0 rz 128.94 deg; joints [131.092, -18.803, 29.508, -102.024, 42.223, 137.009, 25, -128.941]
  MoveL 1191 to (-94.83, -82.94, 83.28) mm, rotated rx 122.81 ry 0 rz 130.36 deg; joints [130.719, -19.19, 30.078, -102.378, 41.903, 138.621, 25, -130.357]
  MoveL 1192 to (-95.14, -84.13, 81.72) mm, rotated rx 122.81 ry 0 rz 130.36 deg; joints [130.656, -19.211, 30.129, -102.437, 41.849, 138.685, 25, -130.357]
  MoveL 1193 to (-96.01, -84.33, 80.49) mm, rotated rx 122.72 ry 0 rz 130.35 deg; joints [130.61, -19.283, 30.225, -102.484, 41.81, 138.82, 25, -130.352]
  MoveL 1194 to (-97.1, -84.13, 79.37) mm, rotated rx 122.23 ry 0 rz 129.97 deg; joints [130.459, -19.436, 30.457, -102.634, 41.683, 139.481, 25, -129.972]
  MoveL 1195 to (-97.66, -84.48, 78.29) mm, rotated rx 121.34 ry 0 rz 129.76 deg; joints [130.208, -19.664, 30.818, -102.89, 41.472, 140.644, 25, -129.759]
  MoveL 1196 to (-97.72, -84.46, 78.24) mm, rotated rx 120.36 ry 0 rz 130.33 deg; joints [130.008, -19.944, 31.215, -103.108, 41.307, 141.857, 25, -130.33]
  MoveL 1197 to (-96.72, -86.5, 77.27) mm, rotated rx 119.93 ry 0 rz 131.3 deg; joints [129.877, -20.072, 31.416, -103.248, 41.199, 142.444, 25, -131.304]
  MoveL 1198 to (-94.59, -89.92, 75.98) mm, rotated rx 119.32 ry 0 rz 133.17 deg; joints [129.702, -20.259, 31.706, -103.444, 41.055, 143.271, 25, -133.168]
  MoveL 1199 to (-93.53, -90.67, 76.38) mm, rotated rx 119.49 ry 0 rz 134.46 deg; joints [129.795, -20.272, 31.672, -103.348, 41.133, 143.001, 25, -134.463]
  MoveL 1200 to (-93.49, -90.71, 76.38) mm, rotated rx 120.86 ry 0 rz 135.09 deg; joints [130.155, -20.004, 31.204, -102.964, 41.432, 141.208, 25, -135.087]
  MoveL 1201 to (-93.61, -86.15, 81.38) mm, rotated rx 123.07 ry 0 rz 133.61 deg; joints [130.827, -19.328, 30.173, -102.286, 41.997, 138.259, 25, -133.608]
  MoveL 1202 to (-93.02, -85.01, 83.24) mm, rotated rx 124.19 ry 0 rz 133.13 deg; joints [131.133, -18.972, 29.665, -101.995, 42.26, 136.827, 25, -133.133]
  MoveL 1203 to (-93.16, -83.79, 84.31) mm, rotated rx 124.24 ry 0 rz 133.05 deg; joints [131.198, -18.954, 29.619, -101.938, 42.316, 136.712, 25, -133.052]
  MoveL 1204 to (-92.9, -82.93, 85.42) mm, rotated rx 124.75 ry 0 rz 132.85 deg; joints [131.353, -18.791, 29.384, -101.797, 42.45, 136.052, 25, -132.845]
  MoveL 1205 to (-94.31, -77.17, 89.2) mm, rotated rx 126.91 ry 0 rz 130.09 deg; joints [131.966, -18.087, 28.409, -101.269, 42.987, 133.33, 25, -130.086]
  Set speed (16.7 mm/s)
  MoveL 1206 to (-106.55, -87.47, 101.21) mm, rotated rx 126.91 ry 0 rz 130.09 deg; joints [131.702, -18.429, 28.035, -100.608, 42.596, 132.367, 25, -130.086]
  Set speed (1000.0 mm/s)
  MoveL 1207 to (-103.93, -86.25, 104.91) mm, rotated rx 127.08 ry 0 rz 130.12 deg; joints [131.841, -18.234, 27.784, -100.497, 42.72, 132.078, 25, -130.12]
  Set speed (5.0 mm/s)
  MoveL 1208 to (-91.73, -75.97, 92.86) mm, rotated rx 127.08 ry 0 rz 130.12 deg; joints [132.102, -17.894, 28.16, -101.157, 43.108, 133.04, 25, -130.12]
  Set speed (16.7 mm/s)
  MoveL 1209 to (-103.58, -86.48, 105.05) mm, rotated rx 127.14 ry 0 rz 130.29 deg; joints [131.86, -18.213, 27.755, -100.482, 42.738, 132.001, 25, -130.292]
  Set speed (1000.0 mm/s)
  MoveL 1210 to (19.02, -119.65, 120.7) mm, rotated rx 135.48 ry 0 rz -171.82 deg; joints [134.303, -15.168, 23.944, -98.885, 44.986, 121.985, 25, -188.183]
  Set speed (5.0 mm/s)
  MoveL 1211 to (17.02, -105.77, 106.44) mm, rotated rx 135.48 ry 0 rz -171.82 deg; joints [134.475, -14.918, 24.42, -99.544, 45.27, 122.956, 25, -188.183]
  Set speed (16.7 mm/s)
  MoveL 1212 to (14.76, -107.9, 104.63) mm, rotated rx 134.52 ry 0 rz -173.14 deg; joints [134.189, -15.275, 24.848, -99.708, 45.004, 124.077, 25, -186.856]
  MoveL 1213 to (14.43, -108.18, 104.38) mm, rotated rx 134.41 ry 0 rz -173.31 deg; joints [134.156, -15.319, 24.901, -99.727, 44.973, 124.207, 25, -186.694]
  MoveL 1214 to (12.82, -109.35, 103.37) mm, rotated rx 133.94 ry 0 rz -174.13 deg; joints [134.013, -15.505, 25.124, -99.813, 44.841, 124.771, 25, -185.869]
  MoveL 1215 to (10.78, -109.97, 102.95) mm, rotated rx 133.95 ry 0 rz -174.17 deg; joints [134.054, -15.586, 25.193, -99.788, 44.878, 124.73, 25, -185.833]
  MoveL 1216 to (9.53, -109.72, 103.33) mm, rotated rx 133.96 ry 0 rz -174.19 deg; joints [134.098, -15.607, 25.202, -99.76, 44.92, 124.693, 25, -185.811]
  MoveL 1217 to (8.48, -108.78, 104.41) mm, rotated rx 133.97 ry 0 rz -174.22 deg; joints [134.16, -15.589, 25.167, -99.723, 44.977, 124.643, 25, -185.782]
  MoveL 1218 to (8.74, -107.31, 105.9) mm, rotated rx 133.99 ry 0 rz -174.25 deg; joints [134.202, -15.507, 25.074, -99.698, 45.016, 124.603, 25, -185.747]
  MoveL 1219 to (9.83, -105.96, 107.16) mm, rotated rx 134.67 ry 0 rz -173.59 deg; joints [134.405, -15.256, 24.771, -99.58, 45.204, 123.806, 25, -186.407]
  MoveL 1220 to (10.74, -103.69, 109.27) mm, rotated rx 136.02 ry 0 rz -172.81 deg; joints [134.803, -14.773, 24.195, -99.36, 45.576, 122.234, 25, -187.195]
  MoveL 1221 to (10.56, -101.91, 110.95) mm, rotated rx 137.24 ry 0 rz -172.69 deg; joints [135.153, -14.336, 23.683, -99.177, 45.905, 120.829, 25, -187.31]
  Set speed (16.7 mm/s)
  MoveL 1222 to (12.28, -115.38, 125.63) mm, rotated rx 137.24 ry 0 rz -172.69 deg; joints [134.999, -14.565, 23.187, -98.526, 45.643, 119.86, 25, -187.31]
  Set speed (1000.0 mm/s)
  MoveL 1223 to (17.45, -114.14, 126.15) mm, rotated rx 137.29 ry 0 rz -172.49 deg; joints [134.905, -14.367, 23.014, -98.579, 45.555, 119.869, 25, -187.505]
  Set speed (5.0 mm/s)
  MoveL 1224 to (15.68, -100.69, 111.46) mm, rotated rx 137.29 ry 0 rz -172.49 deg; joints [135.059, -14.138, 23.511, -99.232, 45.817, 120.838, 25, -187.505]
  Set speed (16.7 mm/s)
  MoveL 1225 to (17.41, -103.52, 108.57) mm, rotated rx 135.68 ry 0 rz -171.76 deg; joints [134.582, -14.746, 24.223, -99.485, 45.37, 122.695, 25, -188.243]
  Set speed (16.7 mm/s)
  MoveL 1226 to (19.41, -117.35, 122.88) mm, rotated rx 135.68 ry 0 rz -171.76 deg; joints [134.412, -14.993, 23.745, -98.828, 45.089, 121.724, 25, -188.243]
  Set speed (1000.0 mm/s)
  MoveL 1227 to (111.82, -88.61, 94.29) mm, rotated rx 124.07 ry 0 rz -127.71 deg; joints [130.807, -19.384, 29.381, -101.368, 41.805, 136.024, 25, -232.292]
  Set speed (5.0 mm/s)
  MoveL 1228 to (98.71, -78.48, 83.09) mm, rotated rx 124.07 ry 0 rz -127.71 deg; joints [131.104, -19.012, 29.72, -102.023, 42.235, 136.976, 25, -232.292]
  Set speed (16.7 mm/s)
  MoveL 1229 to (95.71, -79.78, 85.34) mm, rotated rx 125.1 ry 0 rz -129.02 deg; joints [131.416, -18.683, 29.245, -101.739, 42.505, 135.644, 25, -230.978]
  MoveL 1230 to (94.31, -79.63, 87.01) mm, rotated rx 125.1 ry 0 rz -129.02 deg; joints [131.486, -18.657, 29.189, -101.679, 42.566, 135.581, 25, -230.978]
  MoveL 1231 to (93.97, -78.83, 88.11) mm, rotated rx 125.19 ry 0 rz -129.01 deg; joints [131.53, -18.584, 29.096, -101.639, 42.605, 135.449, 25, -230.989]
  MoveL 1232 to (93.9, -77.73, 89.14) mm, rotated rx 125.67 ry 0 rz -128.63 deg; joints [131.678, -18.426, 28.872, -101.511, 42.734, 134.826, 25, -231.37]
  MoveL 1233 to (93.88, -77.81, 89.09) mm, rotated rx 126.51 ry 0 rz -128.56 deg; joints [131.883, -18.218, 28.577, -101.339, 42.914, 133.806, 25, -231.438]
  MoveL 1234 to (92.11, -77.64, 91.07) mm, rotated rx 127.44 ry 0 rz -129.02 deg; joints [132.167, -17.905, 28.147, -101.107, 43.166, 132.625, 25, -230.978]
  MoveL 1235 to (91.71, -77.52, 91.58) mm, rotated rx 127.44 ry 0 rz -129.02 deg; joints [132.187, -17.893, 28.127, -101.091, 43.183, 132.608, 25, -230.978]
  MoveL 1236 to (91.21, -76.9, 92.59) mm, rotated rx 127.46 ry 0 rz -129.02 deg; joints [132.22, -17.846, 28.067, -101.065, 43.212, 132.557, 25, -230.975]
  MoveL 1237 to (91.08, -75.99, 93.47) mm, rotated rx 127.6 ry 0 rz -128.96 deg; joints [132.268, -17.762, 27.963, -101.026, 43.255, 132.379, 25, -231.045]
  MoveL 1238 to (91.83, -74.28, 94.11) mm, rotated rx 127.6 ry 0 rz -128.96 deg; joints [132.242, -17.676, 27.885, -101.044, 43.231, 132.397, 25, -231.045]
  MoveL 1239 to (92.82, -73.23, 93.96) mm, rotated rx 127.6 ry 0 rz -128.74 deg; joints [132.213, -17.646, 27.865, -101.065, 43.205, 132.417, 25, -231.262]
  MoveL 1240 to (98.07, -69, 91.8) mm, rotated rx 126.56 ry 0 rz -125.58 deg; joints [131.897, -17.996, 28.343, -101.321, 42.925, 133.731, 25, -234.421]
  MoveL 1241 to (98.89, -68.19, 91.53) mm, rotated rx 126.5 ry 0 rz -125.22 deg; joints [131.865, -18.008, 28.368, -101.347, 42.897, 133.817, 25, -234.785]
  MoveL 1242 to (101.69, -66.18, 89.92) mm, rotated rx 125.74 ry 0 rz -123.67 deg; joints [131.632, -18.261, 28.721, -101.544, 42.692, 134.794, 25, -236.327]
  MoveL 1243 to (103.03, -65.73, 88.72) mm, rotated rx 125.71 ry 0 rz -123.69 deg; joints [131.561, -18.265, 28.754, -101.603, 42.63, 134.881, 25, -236.31]
  MoveL 1244 to (103.68, -66.1, 87.68) mm, rotated rx 125.69 ry 0 rz -123.7 deg; joints [131.523, -18.3, 28.806, -101.635, 42.597, 134.933, 25, -236.298]
  MoveL 1245 to (103.76, -67.85, 86.24) mm, rotated rx 125.66 ry 0 rz -123.72 deg; joints [131.506, -18.404, 28.919, -101.653, 42.582, 134.983, 25, -236.277]
  MoveL 1246 to (103.3, -69.35, 85.59) mm, rotated rx 125.36 ry 0 rz -124.42 deg; joints [131.415, -18.502, 29.058, -101.733, 42.503, 135.37, 25, -235.583]
  MoveL 1247 to (103.11, -71.12, 84.37) mm, rotated rx 124.67 ry 0 rz -125.36 deg; joints [131.2, -18.698, 29.352, -101.925, 42.316, 136.269, 25, -234.638]
  Set speed (16.7 mm/s)
  MoveL 1248 to (116.52, -80.64, 95.75) mm, rotated rx 124.67 ry 0 rz -125.36 deg; joints [130.911, -19.064, 29.006, -101.268, 41.894, 135.314, 25, -234.638]
  Set speed (1000.0 mm/s)
  MoveL 1249 to (114.8, -107.23, 67.61) mm, rotated rx 113.91 ry 0 rz -132.44 deg; joints [127.646, -22.377, 34.248, -104.932, 39.207, 150.078, 25, -227.557]
  Set speed (5.0 mm/s)
  MoveL 1250 to (101.3, -94.89, 59.5) mm, rotated rx 113.91 ry 0 rz -132.44 deg; joints [128.06, -21.906, 34.459, -105.514, 39.777, 150.946, 25, -227.557]
  Set speed (16.7 mm/s)
  MoveL 1251 to (98.73, -96.19, 61.7) mm, rotated rx 114.82 ry 0 rz -133.56 deg; joints [128.326, -21.677, 34.035, -105.15, 39.975, 149.638, 25, -226.441]
  MoveL 1252 to (98.26, -96.39, 62.13) mm, rotated rx 114.95 ry 0 rz -133.7 deg; joints [128.37, -21.647, 33.973, -105.09, 40.009, 149.443, 25, -226.305]
  MoveL 1253 to (95.88, -97.29, 64.41) mm, rotated rx 115.89 ry 0 rz -134.64 deg; joints [128.648, -21.403, 33.536, -104.725, 40.221, 148.108, 25, -225.36]
  MoveL 1254 to (94.8, -97.08, 66.3) mm, rotated rx 115.89 ry 0 rz -134.64 deg; joints [128.714, -21.382, 33.473, -104.645, 40.273, 148.021, 25, -225.36]
  MoveL 1255 to (94.8, -96.05, 67.78) mm, rotated rx 116.01 ry 0 rz -134.62 deg; joints [128.764, -21.295, 33.348, -104.576, 40.311, 147.823, 25, -225.383]
  MoveL 1256 to (95.87, -92.99, 70.48) mm, rotated rx 117.16 ry 0 rz -133.36 deg; joints [129.108, -20.982, 32.808, -104.149, 40.58, 146.199, 25, -226.643]
  MoveL 1257 to (96.02, -92.6, 70.8) mm, rotated rx 117.27 ry 0 rz -133.23 deg; joints [129.139, -20.948, 32.753, -104.111, 40.605, 146.053, 25, -226.769]
  MoveL 1258 to (97.67, -89.01, 73.11) mm, rotated rx 118.18 ry 0 rz -131.73 deg; joints [129.409, -20.678, 32.312, -103.789, 40.82, 144.792, 25, -228.269]
  MoveL 1259 to (98.21, -88.1, 73.48) mm, rotated rx 118.18 ry 0 rz -131.73 deg; joints [129.393, -20.63, 32.268, -103.802, 40.806, 144.806, 25, -228.269]
  MoveL 1260 to (98.6, -87.61, 73.56) mm, rotated rx 118.21 ry 0 rz -131.46 deg; joints [129.404, -20.619, 32.251, -103.789, 40.815, 144.755, 25, -228.54]
  MoveL 1261 to (101.35, -84.17, 73.8) mm, rotated rx 118.31 ry 0 rz -129.64 deg; joints [129.429, -20.582, 32.198, -103.76, 40.835, 144.624, 25, -230.356]
  MoveL 1262 to (101.34, -84.09, 73.92) mm, rotated rx 118.79 ry 0 rz -128.78 deg; joints [129.593, -20.545, 32.07, -103.581, 40.97, 143.953, 25, -231.223]
  MoveL 1263 to (101.4, -82.67, 75.44) mm, rotated rx 119.45 ry 0 rz -128.28 deg; joints [129.792, -20.354, 31.76, -103.356, 41.132, 143.043, 25, -231.722]
  MoveL 1264 to (101.61, -81.77, 76.13) mm, rotated rx 119.45 ry 0 rz -128.28 deg; joints [129.791, -20.304, 31.707, -103.354, 41.13, 143.04, 25, -231.722]
  MoveL 1265 to (102.31, -80.38, 76.63) mm, rotated rx 120.21 ry 0 rz -127.11 deg; joints [130.013, -20.157, 31.438, -103.117, 41.314, 142.027, 25, -232.891]
  MoveL 1266 to (101.66, -78.53, 79.4) mm, rotated rx 121.97 ry 0 rz -126.61 deg; joints [130.513, -19.662, 30.67, -102.596, 41.731, 139.694, 25, -233.39]
  MoveL 1267 to (99.3, -78.11, 82.72) mm, rotated rx 123.47 ry 0 rz -127.1 deg; joints [130.966, -19.198, 29.975, -102.154, 42.117, 137.722, 25, -232.904]
  Set speed (16.7 mm/s)
  MoveL 1268 to (112.61, -88.17, 93.75) mm, rotated rx 123.47 ry 0 rz -127.1 deg; joints [130.663, -19.576, 29.643, -101.502, 41.68, 136.773, 25, -232.904]
  Set speed (1000.0 mm/s)
  MoveL 1269 to (116.23, -82.13, 94.81) mm, rotated rx 123.04 ry 0 rz -125.91 deg; joints [130.49, -19.501, 29.643, -101.653, 41.528, 137.361, 25, -234.091]
  Set speed (5.0 mm/s)
  MoveL 1270 to (102.65, -72.3, 83.9) mm, rotated rx 123.04 ry 0 rz -125.91 deg; joints [130.797, -19.119, 29.969, -102.303, 41.97, 138.307, 25, -234.091]
  Set speed (16.7 mm/s)
  MoveL 1271 to (106.23, -70.25, 81.17) mm, rotated rx 121.79 ry 0 rz -124.21 deg; joints [130.42, -19.504, 30.548, -102.675, 41.65, 139.957, 25, -235.787]
  MoveL 1272 to (107.41, -70.03, 79.78) mm, rotated rx 121.79 ry 0 rz -124.21 deg; joints [130.359, -19.513, 30.586, -102.734, 41.598, 140.02, 25, -235.787]
  MoveL 1273 to (107.81, -70.26, 79.04) mm, rotated rx 121.68 ry 0 rz -124.2 deg; joints [130.311, -19.561, 30.659, -102.783, 41.558, 140.183, 25, -235.8]
  MoveL 1274 to (108.44, -71.07, 77.43) mm, rotated rx 120.43 ry 0 rz -124.23 deg; joints [129.972, -19.912, 31.198, -103.141, 41.276, 141.832, 25, -235.77]
  MoveL 1275 to (109.35, -70.9, 76.31) mm, rotated rx 119.93 ry 0 rz -123.94 deg; joints [129.823, -20.057, 31.428, -103.303, 41.153, 142.502, 25, -236.055]
  MoveL 1276 to (109.83, -70.87, 75.65) mm, rotated rx 119.74 ry 0 rz -123.86 deg; joints [129.756, -20.115, 31.524, -103.376, 41.098, 142.773, 25, -236.136]
  MoveL 1277 to (112.42, -70.9, 71.71) mm, rotated rx 118.07 ry 0 rz -123.27 deg; joints [129.251, -20.593, 32.308, -103.955, 40.69, 145.076, 25, -236.734]
  MoveL 1278 to (112.82, -71.03, 70.95) mm, rotated rx 118.07 ry 0 rz -123.27 deg; joints [129.227, -20.609, 32.337, -103.982, 40.67, 145.106, 25, -236.734]
  MoveL 1279 to (113.05, -72.18, 69.4) mm, rotated rx 118.07 ry 0 rz -123.27 deg; joints [129.205, -20.681, 32.427, -104.012, 40.654, 145.14, 25, -236.734]
  MoveL 1280 to (112.94, -72.8, 68.95) mm, rotated rx 117.88 ry 0 rz -123.51 deg; joints [129.149, -20.734, 32.516, -104.081, 40.609, 145.406, 25, -236.489]
  MoveL 1281 to (112.56, -73.82, 68.46) mm, rotated rx 117.88 ry 0 rz -123.51 deg; joints [129.161, -20.787, 32.566, -104.071, 40.62, 145.397, 25, -236.489]
